(* CODESYS project sql_v_2_5_9.library
   DefaultNamespace: Teknike_SQL
   DocFormat: reStructuredText
   Description: Bliblioteca para controle do SQL usando todas as outras blibliotecas
   Author: Tiago B. Cunico
   Title: SQL
   Version: 2.5.9
   Company: Teknike
   Placeholder: Teknike_SQL

Project tree, tasks and I/O mapping:
  libraries: OSCAT - AixOCAT, * (RWTH Aachen University - E.ON Energy Research Center); Tc2_ModbusRTU, * (Beckhoff Automation GmbH); Tc2_Standard, * (Beckhoff Automation GmbH); Tc2_System, * (Beckhoff Automation GmbH); Tc2_Utilities, * (Beckhoff Automation GmbH); Tc3_Database, * (Beckhoff Automation GmbH); Tc3_Module, * (Beckhoff Automation GmbH); Geral, * (Teknike); Partidas, * (Teknike); Sensores, * (Teknike)
  FBs/
    Emergencias/
      function block FB_CriaTabelaEmergencias [ST]: GeraAsEmergencias, GeraTabela
      function block FB_IniciaOsBlocosDaEmergencia [ST]
    Grupos/
      Sts/
        data type ST_BancoGrupo
        data type st_ConfigGrupo
        data type st_EntradaGrupo
        data type st_Grupo
        data type st_SaidaGrupo
      function F_StringSeparadorFBGrupos [ST]
      function block FB_ControleGrupo [ST]: AjustaEntrada, AjustaSaida, GeraTabela, MaquinaDeEstado
      function block FB_IniciaGrupos [ST]: GeraOsGrupos, GeraTabela, MaquinaInica
    IHM/
      STs/
        data type st_OutrosInterlocks
      function block FB_GeraListaInterlocksIHM [ST]
    Iluminacao/
      Duts/
        data type ConfigTelerruptorDB
        data type enum_GravaNomes
        data type enum_LeituradosNomes
      function block FB_ConfigDoTelerruptor [ST]: GeraOsTelerruptores, GeraTabela, GravaValores, LeNomes
    Intralogistica/
      Top10SKU/
        data type DUT_Top10SKU
        data type Enum_HistorogramaSKUs
        function block FB_HistogramaSKUsMaisLidas [ST]: Evento, GeraTabela, Tabela, Top10
        TODO.txt
    MedicaoEnergia/
      Duts/
        PM2100_485_Schneider/
          data type config_PM2100_485_Schneider
          data type entrada_PM2100_485_Schneider
          data type saida_PM2100_485_Schneider
          data type st_PM2100_485_Schneider
          data type State_Modbus
          data type stCorrente
          data type stDemanda
          data type stEnergia
          data type stPotencia
          data type stTensao
        SEPAMS20_485_Schneider/
          data type config_SEPAMS20_Schneider
          data type entrada_SEPAMS20_Schneider
          data type saida_SEPAMS20_Schneider
          data type st_SEPAMS20_Schneider
          data type stCorrenteSEPAM
          data type stTemposSEPAM
          data type stTensaoSEPAM
        data type stCentroDeCusto
        data type stConfigNomeMedidorDB
        data type stCorrenteCSV
        data type stEscreveNoSQL
        data type stLeDoSQL
        data type stMedia15min
        data type stMediaAno
        data type stMediaDia
        data type stMediaMes
        data type stMinuto
        data type stOrganizaDados
      function block FB_CentroDeCustos2 [ST]: LeValores
      function block FB_DBCentroDeCustos [ST]: DeleteValores, GeraTabela, GravaValores, LeValores
      function block FB_DBMedidores [ST]: GeraTabela, GravaValores, LeValores
      function block FB_LeBancoDeDadosParaCSV [ST]: GeraTabela, LeValores
      function block FB_NomesMedidoresPM2100 [ST]: GeraOsMedidores, GeraTabela, GravaValores, LeNomes
      function block FB_NomesMedidoresSEPAM [ST]: GeraOsMedidores, GeraTabela, GravaValores, LeNomes
      function block FB_SalvaDadosMedidores [ST]: GeraTabela, GravaValores
    Partidas/
      KPI/
        function block FB_KPIPartidasSQL [ST]: GeraTabela, GravaHistorico
        data type st_KPISQL
      SalvaUsoNormal/
        function block FB_BDMotores [ST]: AtualizaValor, EscreveCSV, GeraTabela
        data type st_EscritaBD
      st/
        data type enum_MaquinaConfigPartidaDB
        data type st_LeConfigPartidaNoBanco_1
      function block FB_ConfigPartidaNoBanco [ST]: CalculaEmergencia, CalculaInterlock, ExecutaEstadoLeitura, GeraEmergencias, GeraNomeInterlock, LinkaOsNaoInterlock, MudouNoMotor, TrocaEstadoLeitura, ZeraReferencias
      function block FB_CriaTabelaEMotoresParaInterlock [ST]: GeraOsMotores, GeraTabela
      function block FB_IniciaOsBlocosDeConfigDoMotor [ST]: AtualizaTagEmergencias, AtualizaTagInterlocks, LinkaOsNaoInterlocks
    Sensores/
      fb_Hidrometro/
        dut/
          data type st_Hidrometro
        function block FB_Hidrometro [ST]: SalvaHistorico
      St/
        data type st_ComparaAnalogico
        data type st_LeComparaAnalogico
      function block FB_AtualizaTag [ST]: Atualiza, GeraTabela
      function block FB_CriaTabelaSensores [ST]: GeraOsSensores, GeraTabela
      function block FB_DBComparaSensor [ST]: GeraTabela, GravaValores
      function block FB_HistoricoSQL [ST]: GeraTabela, GravaHistorico
      function block FB_HistoricoTag [ST]: Atualiza, GeraTabela
      function block FB_IniciaOsBlocosDeSensor [ST]
    Valvula/
      BancoValvula/
  00000000-0000-0000-0000-000000000000|FBs\Intralogistica\Top10SKU\TODO.txt
  POUs/
    global variables GVL_BlibliotecaSQL
    program MAIN [ST]
    program ValidaLicensa [ST]: Licensas
  Project Information/
    function F_GetCompany [ST]
    function F_GetTitle [ST]
    function F_GetVersion [ST]
  Version/
    global variables Global_Version
  VISUs/
*)

// FBs/Grupos/Sts/ST_BancoGrupo
TYPE ST_BancoGrupo :
STRUCT
	ID: LINT;
	Nome: STRING(80);
	Motores: STRING(255);
	Timestamp: DT;
END_STRUCT
END_TYPE

// FBs/Grupos/Sts/st_ConfigGrupo
TYPE st_ConfigGrupo :
STRUCT PERSISTENT RETAIN
	sMotores: STRING(255);//se ele nao conseguir ler do banco ele pega daqui
	sNome : STRING;
	xCascata : BOOL;// assim ele usa cascata
	rTempoCascata : REAL; // ignora se a partida diz que ta show e liga por esse tempo
	xInterDependependes : BOOL; // se uma parar para todas
END_STRUCT
END_TYPE

// FBs/Grupos/Sts/st_EntradaGrupo
TYPE st_EntradaGrupo :
STRUCT
	xLiga : BOOL;
	xLigaFisico : BOOL;
	xReset : BOOL;
END_STRUCT
END_TYPE

// FBs/Grupos/Sts/st_Grupo
TYPE st_Grupo :
STRUCT
	En : st_EntradaGrupo;
	Sa : st_SaidaGrupo;
	Config : st_ConfigGrupo;
	Banco : ST_BancoGrupo;
END_STRUCT
END_TYPE

// FBs/Grupos/Sts/st_SaidaGrupo
TYPE st_SaidaGrupo :
STRUCT
	xError : BOOL;
	xInterlock : BOOL;
	xEmergencia : BOOL;
	xLigado : BOOL;
	xLigando : BOOL;
	sStatus : STRING;
	sStatusPartidas : ARRAY[0..100] OF STRING;
END_STRUCT
END_TYPE

// FBs/IHM/STs/st_OutrosInterlocks
TYPE st_OutrosInterlocks :
	STRUCT
		sTag	: STRING;
		xEstado	: BOOL;
	END_STRUCT
END_TYPE

// FBs/Iluminacao/Duts/ConfigTelerruptorDB
TYPE ConfigTelerruptorDB :
STRUCT
	Telerruptor: DINT;
	Tag: STRING(80);
	Funcao: STRING(80);
END_STRUCT
END_TYPE

// FBs/Iluminacao/Duts/enum_GravaNomes
{attribute 'qualified_only'}
{attribute 'strict'}
TYPE enum_GravaNomes :
(
	eEsperando := 0,
	eAbreConexao := 1,
	eGravaNomes := 2,
	eCriaComando := 3,
	eFechaConexao := 4,
	eParado := 100
);
END_TYPE

// FBs/Iluminacao/Duts/enum_LeituradosNomes
{attribute 'qualified_only'}
{attribute 'strict'}
TYPE enum_LeituradosNomes :
(
	eEsperando := 0,
	eAbreConexao := 1,
	eLeOsNomes := 2,
	eMonitoraTrocaDeNomes := 3,
	eFechaConexao := 4,
	eParado := 100
);
END_TYPE

// FBs/Intralogistica/Top10SKU/DUT_Top10SKU
TYPE DUT_Top10SKU :
STRUCT
	SKU : LINT;
	Contagem : LINT;
END_STRUCT
END_TYPE

// FBs/Intralogistica/Top10SKU/Enum_HistorogramaSKUs
{attribute 'qualified_only'}
//{attribute 'strict'}
TYPE Enum_HistorogramaSKUs :
(
	erro := 0,
	Esperando,
	AbreConexao,
	CriaComando,
	Grava,
	DeletaEvento,
	CriaEvento,
	Vetop10,
	FechaConexao
);
END_TYPE

// FBs/MedicaoEnergia/Duts/PM2100_485_Schneider/config_PM2100_485_Schneider
TYPE config_PM2100_485_Schneider :
STRUCT PERSISTENT RETAIN
	iEndereco 			: INT;
	sNomeFuncao			: STRING; 
END_STRUCT
END_TYPE

// FBs/MedicaoEnergia/Duts/PM2100_485_Schneider/entrada_PM2100_485_Schneider
TYPE entrada_PM2100_485_Schneider :
STRUCT
	xInicia				: BOOL; //Inicia a leitura
	xAtualizaCorrente	: BOOL := TRUE; //Habilita para ler os parametros de corrente
	xAtualizaTensao		: BOOL;	//Habilita para ler os parametros de tensao
	xAtualizaPotencia	: BOOL; //Habilita para ler os parametros de potencia
	xAtualizaEnergia	: BOOL := TRUE; //Habilita para ler os parametros de energia
	xAtualizaDemanda	: BOOL := TRUE; //Habilita para ler os parametros de demanda
END_STRUCT
END_TYPE

// FBs/MedicaoEnergia/Duts/PM2100_485_Schneider/saida_PM2100_485_Schneider
TYPE saida_PM2100_485_Schneider :
STRUCT
	xTerminei					: BOOL;	
	xOnline						: BOOL;
	UltimoModbusErro			: ST_ModbusErrorDiagnostics;
	sStatus						: STRING;
	Corrente: stCorrente;
	Tensao	: stTensao;
	Energia	: stEnergia;
	Potencia: stPotencia;
	Demanda	: stDemanda;
END_STRUCT
END_TYPE

// FBs/MedicaoEnergia/Duts/PM2100_485_Schneider/st_PM2100_485_Schneider
TYPE st_PM2100_485_Schneider :
STRUCT
	en		: entrada_PM2100_485_Schneider;
	sa		: saida_PM2100_485_Schneider;
	config	: config_PM2100_485_Schneider;
END_STRUCT
END_TYPE

// FBs/MedicaoEnergia/Duts/PM2100_485_Schneider/State_Modbus
{attribute 'qualified_only'}
{attribute 'strict'}
TYPE State_Modbus :
(
	Inicia			:= 0,
	LeituraCorrente	:= 1,
	LeituraTensao	:= 2,
	LeituraPotencia	:= 3,
	LeituraEnergia	:= 4,
	LeituraDemanda	:= 5,
	LeituraTempos	:= 6 
);
END_TYPE

// FBs/MedicaoEnergia/Duts/PM2100_485_Schneider/stCorrente
TYPE stCorrente :
STRUCT
	//Corrente
	rCorrenteA		: REAL;
	rCorrenteB		: REAL;
	rCorrenteC		: REAL;
	rCorrenteMedia	: REAL;
END_STRUCT
END_TYPE

// FBs/MedicaoEnergia/Duts/PM2100_485_Schneider/stDemanda
TYPE stDemanda :
STRUCT
	//Demanda
	rDemandaDePotenciaAtiva		: REAL;
	rDemandaDePotenciaReativa	: REAL;
	rDemandaDePotenciaAparente	: REAL;
END_STRUCT
END_TYPE

// FBs/MedicaoEnergia/Duts/PM2100_485_Schneider/stEnergia
TYPE stEnergia :
STRUCT
	//Energia
	rPotenciaAtivaEntregue		: REAL;
	rPotenciaAtivaRecebida		: REAL;
	rPotenciaReativaEntregue	: REAL;
	rPotenciaReativaRecebida	: REAL;
	rPotenciaAparenteEntregue	: REAL;
	rPotenciaAparenteRecebida	: REAL;
END_STRUCT
END_TYPE

// FBs/MedicaoEnergia/Duts/PM2100_485_Schneider/stPotencia
TYPE stPotencia :
STRUCT
	//Potencia
	rPotenciaAtivaTotal		: REAL;
	rPotenciaReativaTotal	: REAL;
	rPotenciaAparenteTotal	: REAL;
	rFatorDePotenciaTotal	: REAL;
END_STRUCT
END_TYPE

// FBs/MedicaoEnergia/Duts/PM2100_485_Schneider/stTensao
TYPE stTensao :
STRUCT
	//Tensao
	rTensaoAN		: REAL;
	rTensaoBN		: REAL;
	rTensaoCN		: REAL;
	rTensaoMediaLN	: REAL;
	rTensaoAB		: REAL;
	rTensaoBC		: REAL;
	rTensaoAC		: REAL;
	rTensaoMediaLL	: REAL;
END_STRUCT
END_TYPE

// FBs/MedicaoEnergia/Duts/SEPAMS20_485_Schneider/config_SEPAMS20_Schneider
TYPE config_SEPAMS20_Schneider :
STRUCT PERSISTENT RETAIN
	iEndereco 			: INT;
	sNomeFuncao			: STRING;
END_STRUCT
END_TYPE

// FBs/MedicaoEnergia/Duts/SEPAMS20_485_Schneider/entrada_SEPAMS20_Schneider
TYPE entrada_SEPAMS20_Schneider :
STRUCT
	xInicia				: BOOL; //Inicia a leitura
	xAtualizaCorrente	: BOOL := TRUE; //Habilita para ler os parametros de corrente
	xAtualizaTensao		: BOOL := TRUE;	//Habilita para ler os parametros de tensao
	xAtualizaTempos		: BOOL; //Habilita para ler os parametros que indicam tempos de atuação do disjuntor
END_STRUCT
END_TYPE

// FBs/MedicaoEnergia/Duts/SEPAMS20_485_Schneider/saida_SEPAMS20_Schneider
TYPE saida_SEPAMS20_Schneider :
STRUCT
	xTerminei					: BOOL;	
	xOnline						: BOOL;
	UltimoModbusErro			: ST_ModbusErrorDiagnostics;
	sStatus						: STRING;
	
	rDemandaAparente			: REAL;	
	Corrente					: stCorrenteSEPAM;
	Tensao						: stTensaoSEPAM;
	Tempos						: stTemposSEPAM;
END_STRUCT
END_TYPE

// FBs/MedicaoEnergia/Duts/SEPAMS20_485_Schneider/st_SEPAMS20_Schneider
TYPE st_SEPAMS20_Schneider :
STRUCT
	en		: entrada_SEPAMS20_Schneider;
	sa		: saida_SEPAMS20_Schneider;
	config	: config_SEPAMS20_Schneider;
END_STRUCT
END_TYPE

// FBs/MedicaoEnergia/Duts/SEPAMS20_485_Schneider/stCorrenteSEPAM
TYPE stCorrenteSEPAM :
STRUCT
	//Corrente
	rCorrente1		: REAL;
	rCorrente2		: REAL;
	rCorrente3		: REAL;
	rCorrente1Media	: REAL;
	rCorrente2Media	: REAL;
	rCorrente3Media	: REAL;
	rCorrenteTrip1	: REAL;
	rCorrenteTrip2	: REAL;
	rCorrenteTrip3	: REAL;
END_STRUCT
END_TYPE

// FBs/MedicaoEnergia/Duts/SEPAMS20_485_Schneider/stTemposSEPAM
TYPE stTemposSEPAM :
STRUCT
	iTempoDeOperacao					: INT;
	iTempoDeOperacaoAntesDoTrip			: INT;
	iTempoDeEsperaAposTripPorSobrecarga	: INT;
	iTempoDeInibicaoDePartida			: INT;
END_STRUCT
END_TYPE

// FBs/MedicaoEnergia/Duts/SEPAMS20_485_Schneider/stTensaoSEPAM
TYPE stTensaoSEPAM :
STRUCT
	rTensaoV1	: REAL;
	rTensaoV2	: REAL;
	rTensaoV3	: REAL;
	rTensaoU21	: REAL;
	rTensaoU32	: REAL;
	rTensaoU13	: REAL;
END_STRUCT
END_TYPE

// FBs/MedicaoEnergia/Duts/stCentroDeCusto
TYPE stCentroDeCusto :
STRUCT
	NomeGrupo				: STRING(255);
	MedidoresSelecionados	: STRING(255);
	Timestamp				: DT;
END_STRUCT
END_TYPE

// FBs/MedicaoEnergia/Duts/stConfigNomeMedidorDB
TYPE stConfigNomeMedidorDB :
STRUCT
	Medidor: DINT;
	Tag: STRING(80);
	Funcao: STRING(80);
END_STRUCT
END_TYPE

// FBs/MedicaoEnergia/Duts/stCorrenteCSV
TYPE stCorrenteCSV :
STRUCT
	rCorrenteA				: REAL;
	rCorrenteB				: REAL;
	rCorrenteC				: REAL;
	rCorrenteMedia			: REAL;
	Medidor					: INT;
	Timestamp				: DT;
END_STRUCT
END_TYPE

// FBs/MedicaoEnergia/Duts/stEscreveNoSQL
TYPE stEscreveNoSQL :
STRUCT
	rDemanda1min			: REAL;
	rFatorDePotencia1min	: REAL;
	rConsumo1min			: REAL;
	xTrocouMinuto			: BOOL;
END_STRUCT
END_TYPE

// FBs/MedicaoEnergia/Duts/stLeDoSQL
TYPE stLeDoSQL :
STRUCT
	Minuto		: ARRAY[1..15] OF stMinuto;
	Media15min	: ARRAY[1..96] OF stMedia15min;
	MediaDia	: ARRAY[1..31] OF stMediaDia;
	MediaMes	: ARRAY[1..12] OF stMediaMes;
END_STRUCT
END_TYPE

// FBs/MedicaoEnergia/Duts/stMedia15min
TYPE stMedia15min :
STRUCT
	rMedia15min				: REAL;
	rFatorDePotencia15min	: REAL;
	rConsumo15min			: REAL;
	Medidor					: INT;
	Timestamp				: DT;
END_STRUCT
END_TYPE

// FBs/MedicaoEnergia/Duts/stMediaAno
TYPE stMediaAno :
STRUCT
	rMediaAno			: REAL;
	rFatorDePotenciaAno	: REAL;
	rConsumoAno			: REAL;
	Medidor				: INT;
	Timestamp			: DT;
END_STRUCT
END_TYPE

// FBs/MedicaoEnergia/Duts/stMediaDia
TYPE stMediaDia :
STRUCT
	rMediaDia				: REAL;
	rFatorDePotenciaDia		: REAL;
	rConsumoDia				: REAL;
	Medidor					: INT;
	Timestamp				: DT;
END_STRUCT
END_TYPE

// FBs/MedicaoEnergia/Duts/stMediaMes
TYPE stMediaMes :
STRUCT
	rMediaMes			: REAL;
	rFatorDePotenciaMes	: REAL;
	rConsumoMes			: REAL;
	Medidor				: INT;
	Timestamp			: DT;
END_STRUCT
END_TYPE

// FBs/MedicaoEnergia/Duts/stMinuto
TYPE stMinuto :
STRUCT
	rDemanda1min		: REAL;
	rFatorDePotencia1min: REAL;
	rConsumo1min		: REAL;
	Medidor				: INT;
	Timestamp			: DT;
END_STRUCT
END_TYPE

// FBs/MedicaoEnergia/Duts/stOrganizaDados
TYPE stOrganizaDados :
STRUCT
	iMedidor	: INT;
	minuto		: ARRAY[1..15] OF stMinuto;
	media15min	: ARRAY[1..96] OF stMedia15min;
	MediaDia	: ARRAY[1..31] OF stMediaDia;
	MediaMes	: ARRAY[1..12] OF stMediaMes;
END_STRUCT
END_TYPE

// FBs/Partidas/KPI/st_KPISQL
TYPE st_KPISQL :
STRUCT
	ID : T_ULARGE_INTEGER;
	TAG : STRING;
	Desligado : REAL;
	Ligado : REAL;
	Emergencia : REAL;
	Falha : REAL;
	Interlock : REAL;
	//Timestamp : DT;
END_STRUCT
END_TYPE

// FBs/Partidas/SalvaUsoNormal/st_EscritaBD

TYPE st_EscritaBD :
	STRUCT
		ID					: T_ULARGE_INTEGER;
		Velocidade			: INT;
		Corrente			: REAL;
		TemperaturaDoMotor	: REAL;
		Torque				: REAL;
		StatusIHM			: STRING;
		HorimetroD			: STRING;
		TotalDePartidas		: INT;
		TotalDeFalhas		: INT;
	END_STRUCT
END_TYPE

// FBs/Partidas/st/enum_MaquinaConfigPartidaDB
{attribute 'qualified_only'}
{attribute 'strict'}
TYPE enum_MaquinaConfigPartidaDB :
(
	Esperando := 0,
	AbreConexao,
	CriaComando,
	Gravando,
	FechaConexao,
	LendoEleMesmo,
	LinkaOsNaoInterlock,
	ProcuraTag1,
	ProcuraTag2,
	Gera_sInterlock,
	Gera_Emergencia,
	ExecutaInterlocks,
	falha
);
END_TYPE

// FBs/Partidas/st/st_LeConfigPartidaNoBanco_1
TYPE ST_ConfigMotorDB_1 :
	STRUCT
		Motor	: T_ULARGE_INTEGER;
		Tag		: STRING(80);
		Funcao	: STRING(80);

		InvIT1A	: INT;
		IT1A	: STRING(80);
		OPIT1	: INT;
		InvIT1B	: INT;
		IT1B	: STRING(80);

		InvIT2A	: INT;
		IT2A	: STRING(80);
		OPIT2	: INT;
		InvIT2B	: INT;
		IT2B	: STRING(80);

		InvIT3A	: INT;
		IT3A	: STRING(80);
		OPIT3	: INT;
		InvIT3B	: INT;
		IT3B	: STRING(80);

		InvIT4A	: INT;
		IT4A	: STRING(80);
		OPIT4	: INT;
		InvIT4B	: INT;
		IT4B	: STRING(80);
		
		Timestamp : DT;

	END_STRUCT
END_TYPE

// FBs/Sensores/fb_Hidrometro/dut/st_Hidrometro
TYPE st_Hidrometro :
STRUCT
	rContadorTotal : REAL;
	rContadorHoje : REAL;
	xSinal : BOOL;
	xReset : BOOL;
	Historico : ARRAY[0..180] OF st_HistoricoHidrometro;
	rMultiplicadorVazao : REAL := 0.1;
END_STRUCT
END_TYPE

// FBs/Sensores/St/st_ComparaAnalogico
TYPE st_ComparaAnalogico :
STRUCT
	rAnalogicoLido	: REAL;
	rAnalogicoManual: REAL;
	rDiferenca		: REAL;
	xSalva			: BOOL;
END_STRUCT
END_TYPE

// FBs/Sensores/St/st_LeComparaAnalogico
TYPE st_LeComparaAnalogico :
	STRUCT
		Sensor			: T_ULARGE_INTEGER;
		rAnalogicoLido	: REAL;
		rAnlogicoManual	: REAL;
		rDiferenca		: REAL;
		xSalva			: BOOL;
	END_STRUCT
END_TYPE

// POUs/GVL_BlibliotecaSQL
//{attribute 'qualified_only'}
VAR_GLOBAL
    {attribute 'hide'} 
	{attribute 'tc_no_symbol'}
	xLicensaValida651641iih : BOOL;
	LicensaValida : BOOL;
	STCheckLicense : ST_CheckLicense;
END_VAR

// Version/Global_Version
{attribute 'TcGenerated'}
{attribute 'no-analysis'}
{attribute 'linkalways'}
// This function has been automatically generated from the project information.
VAR_GLOBAL CONSTANT
	{attribute 'const_non_replaced'}
	stLibVersion_SQL : ST_LibVersion := (iMajor := 2, iMinor := 5, iBuild := 9, iRevision := 0, nFlags := 0, sVersion := '2.5.9');
END_VAR

// FBs/Emergencias/FB_CriaTabelaEmergencias
(*
	Bloco para gerar a tabela das emergencias de forma generica
*)


{attribute 'hide_all_locals'}
FUNCTION_BLOCK FB_CriaTabelaEmergencias
VAR_IN_OUT
	Emergencias : ARRAY[*] OF st_Emergencia;
END_VAR
VAR_INPUT
	xCriaTabela		: BOOL;
	iNumeroDataBase	: INT		:= 1;
	sNomeDataBase	: STRING	:= 'EmergenciaConfig';
END_VAR
VAR_OUTPUT
	xOcupado : BOOL;
END_VAR
VAR
	i				: INT;
	xGeraMoto		: BOOL;
	diParteBaixa	: DINT;
	diParteAlta		: DINT;

	//Grava valores
	xGravando		: BOOL;
	rtEscrita		: R_TRIG;
	xEscreve		: BOOL;
	EstruturaBanco	: st_Emergencia_Banco;
	xEscreveAux		: BOOL;
	sAux			: ARRAY[1..50] OF STRING(80);
	fbPLCDBWrite	: FB_PLCDBWriteEvt(sNetID := '', tTimeout := T#30S); //Bloco para gravar no banco de dados

	ColumnNamesGrava : ARRAY[0..2] OF STRING(50) := ['Emergencia',
													'Tag',
													'Funcao'];

	//Cria table
	rtCria			: R_TRIG;
	xCria			: BOOL;
	fbPLCDBCreate	: FB_PLCDBCreateEvt(sNetID := '', tTimeout := T#30S);

	ColumnInfo :
		ARRAY[0..3] OF ST_ColumnInfo
		:= [(sName := 'Emergencia', eType := E_ColumnType.BigInt, nLength := 8, sProperty := 'IDENTITY(1,1)'),
				(sName := 'Tag', eType := E_ColumnType.NVarChar, nLength := 80, sProperty := 'DEFAULT $'SEMTAG$''),
				(sName := 'Funcao', eType := E_ColumnType.NVarChar, nLength := 80, sProperty := 'DEFAULT $'NADA$''),
				(
				sName := 'Timestamp',
					eType := E_ColumnType.DateTime,
					nLength := 4,
					sProperty := 'DEFAULT CURRENT_TIMESTAMP ON UPDATE CURRENT_TIMESTAMP')];
END_VAR

IF xLicensaValida651641iih THEN
	GeraTabela();
	GeraAsEmergencias();
END_IF

ACTION GeraAsEmergencias:

diParteBaixa	:= LOWER_BOUND(Emergencias, 1);
diParteAlta		:= UPPER_BOUND(Emergencias, 1);

IF xGeraMoto THEN

	xEscreve := TRUE;
	rtEscrita(CLK := xEscreve, Q =>);

	IF rtEscrita.q THEN
		xEscreveAux						:= TRUE;
		//EstruturaBanco.Sensor.dwLowPart	:= DINT_TO_DWORD(diParteBaixa + i);
		EstruturaBanco.Tag				:= CONCAT('Emer', TO_STRING(i));
	END_IF

	IF xEscreveAux THEN
		IF fbPLCDBWrite.WriteStruct
			(
				hDBID := INT_TO_UDINT(iNumeroDataBase),
					sTableName := sNomeDataBase,
					pRecord := ADR(EstruturaBanco),
					cbRecord := SIZEOF(EstruturaBanco),
					pColumnNames := ADR(ColumnNamesGrava),
					cbColumnNames := SIZEOF(ColumnNamesGrava))
		THEN
			xEscreve := FALSE;
			rtEscrita(CLK := xEscreve, Q =>);
			xEscreveAux	:= FALSE;
			i			:= i + 1;

			IF i > diParteAlta THEN
				xGeraMoto	:= FALSE;
				xOcupado	:= FALSE;
			END_IF
		END_IF
	END_IF

END_IF
END_ACTION

ACTION GeraTabela:

rtCria(CLK := xCriaTabela, Q =>);

IF rtCria.q THEN
	xCria		:= TRUE;
	xOcupado	:= TRUE;
END_IF

IF xCria THEN

	IF fbPLCDBCreate.Table
		(
			hDBID := INT_TO_UDINT(iNumeroDataBase),
				sTableName := sNomeDataBase,
				pTableCfg := ADR(ColumnInfo),
				cbTableCfg := SIZEOF(ColumnInfo))
	THEN
		IF NOT fbPLCDBCreate.bError THEN
			xCria		:= FALSE;
			xCriaTabela	:= FALSE;
			xGeraMoto	:= TRUE;
			i			:= 1;
		ELSE
			xCria		:= FALSE;
			xCriaTabela	:= FALSE;
		END_IF
	END_IF

END_IF
END_ACTION

END_FUNCTION_BLOCK

// FBs/Emergencias/FB_IniciaOsBlocosDaEmergencia
{attribute 'hide_all_locals'}
FUNCTION_BLOCK FB_IniciaOsBlocosDaEmergencia
VAR_IN_OUT
	stEmergencias : ARRAY[*] OF st_Emergencia;
	sPossiveisEmergencias : ARRAY[*] OF STRING;
END_VAR
VAR_INPUT
	xInicia : BOOL;
	iNumeroDataBase	: INT		:= 1;
	sNomeDataBase	: STRING	:= 'EmergenciaConfig';
END_VAR
VAR_OUTPUT
END_VAR
VAR
	fbPLCDBCmd			: FB_PLCDBCmdEvt(sNetID := '', tTimeout := T#60S);
	fbSQLDatabase		: FB_SQLDatabaseEvt(sNetID := '', tTimeout := T#60S);
	sCmd				: STRING(1000);
	sCmdUpdate			: STRING(1000);
	stPara				: ST_ExpParameter;
	TagAProcurar		: STRING(80);
	nRecords			: UDINT;
	xProcuraNaTabela	: BOOL;
	EstruturaBanco		: ARRAY[0..999] OF Teknike_Geral.st_Emergencia_Banco;
	xJogaNoInterlock	: BOOL;
	sTag1				: STRING;
	sTag2				: STRING;
	xEMotor				: BOOL;
	sMensagemErro1		: STRING;
	diCimaSensor		: DINT;
	diBaixoSensor		: DINT;

	iEstado	: INT := 1;
	i		: INT;

	iAux : INT;
	
	EstruturaBancoVazio: Teknike_Geral.st_Emergencia_Banco;

END_VAR


IF xLicensaValida651641iih THEN
	
	
	CASE iEstado OF
		1: //Esperando
			IF xInicia THEN
				iEstado := 2;
			END_IF
	
		2: //abre conexao
			IF fbSqlDatabase.Connect(int_to_udint(iNumeroDataBase)) THEN
				IF fbSqlDatabase.bError THEN
					IF fbSqlDatabase.ipTcResult.ipSourceInfo.sName = 'ADSERR_DEVICE_LICENSENOTFOUND' THEN
						// se der isso ele nao fica tentando e gerando uma caralhada de erro pq nao tem a lisença
						iEstado := 0;
					ELSE
						iEstado := 2;
					END_IF
				ELSE
					IF fbSqlDatabase.bConnected THEN
						iEstado := 3;
					END_IF
				END_IF
			END_IF
	
		3: // le o role
			TagAProcurar		:= sTag1;
			stPara.eParaType	:= E_ExpParameterType.STRING_;
			stPara.nParaSize	:= SIZEOF(TagAProcurar);
			stPara.sParaName	:= 'Tag';
	
			diBaixoSensor	:= LOWER_BOUND(stEmergencias, 1);
			diCimaSensor	:= UPPER_BOUND(stEmergencias, 1);
	
			// set command with placeholder
			sCmd := CONCAT(CONCAT('SELECT * FROM ',sNomeDataBase),';');
	
			// call functionblock
			IF fbPLCDBCmd.ExecuteDataReturn
				(
					hDBID := 1,
						pExpression := ADR(sCmd),
						cbExpression := SIZEOF(sCmd),
						pData := ADR(TagAProcurar),
						cbData := SIZEOF(TagAProcurar),
						pParameter := ADR(stPara),
						cbParameter := SIZEOF(stPara),
						nStartIndex := 0,
						nRecordCount := DINT_TO_UDINT(diCimaSensor-1),
						pReturnData := ADR(EstruturaBanco),
						cbReturnData := SIZEOF(EstruturaBanco),
						pRecords := ADR(nRecords))
			THEN
				IF fbPLCDBCmd.bError THEN
					sMensagemErro1 := 'Nao conseguiu a tag';
				ELSE
					sMensagemErro1	:= 'Conseguiu a tag';
					iEstado			:= 4;
					
					//Fica forçado pra poder ter uma emergencia geral, tipo juntar varias numa
					IF diBaixoSensor = 0 THEN
						stEmergencias[0].Banco.Tag := 'Emergencia Geral';
					END_IF
	
					FOR i := TO_INT(diBaixoSensor) TO TO_INT(diCimaSensor)-1 DO
						stEmergencias[i+1].Banco := EstruturaBanco[i];
					END_FOR
					//Essa aqui fica vazia so pro framework aceitar colocar vazio
					stEmergencias[diCimaSensor].Banco := EstruturaBancoVazio;
				END_IF
			END_IF
	
		4: // FechaConexao conexao
			IF fbSqlDatabase.Disconnect() THEN
	
				xInicia := FALSE;
	
				IF fbSqlDatabase.bError THEN
					iEstado := 1;
				ELSE
					iEstado := 1;
				END_IF
				
				//IF LOWER_BOUND(sPossiveisEmergencias,1) = LOWER_BOUND(stEmergencias,1) AND UPPER_BOUND(sPossiveisEmergencias,1)+1 = UPPER_BOUND(stEmergencias,1) THEN	
					FOR i:= TO_INT(LOWER_BOUND(sPossiveisEmergencias,1)) TO TO_INT(UPPER_BOUND(sPossiveisEmergencias,1)) DO
						sPossiveisEmergencias[i] := stEmergencias[i].Banco.Tag;
					END_FOR
				//ELSE
				//	sPossiveisEmergencias[LOWER_BOUND(sPossiveisEmergencias,1)] := 'Vetor de tamanho errado';
				//END_IF
				
				
			END_IF
	END_CASE

END_IF

END_FUNCTION_BLOCK

// FBs/Grupos/F_StringSeparadorFBGrupos
FUNCTION F_StringSeparadorFBGrupos : BOOL
VAR_INPUT
	sStr : STRING;
END_VAR
VAR_IN_OUT
	ListaINT : ARRAY[*] OF INT;
END_VAR
VAR
	iListIntMIN : INT;
	iListIntMAX : INT;
	
	sParteEsquerda : STRING;
	sResto : STRING;
	sSepara : STRING;
	
	sNumeroInicio : STRING;
	sNumeroFim : STRING;
	
	i: INT;
	j: INT;
	
	iIndex : INT;
END_VAR


iListIntMIN := DINT_TO_INT(LOWER_BOUND(ListaINT,1));
iListIntMAX := DINT_TO_INT(UPPER_BOUND(ListaINT,1));

FOR i:= iListIntMIN TO iListIntMAX DO
	ListaINT[i] := 0;
END_FOR


sSepara := sStr;
iIndex := iListIntMIN;

//O codigo aqui vai pegar a string que a gente guarda no banco de dados e separar onde tem ","
//quando ele separa ele ve se dentro ta um "-", que nesse caso esta servindo para colocar os motores dentro de um periodo
// entao se se ele revceber a string 1-5,7,10 ele devolver na lista os motores do 1,2,3,4,5,7,10
//ele olha tb ser nao entrou um motor 2 vezes, se for o caso ele considera so a primeira vez

WHILE FindAndSplit(
		pSeparator:= ADR(','), 
		pSrcString:= ADR(sSepara), 
		pLeftString:= ADR(sParteEsquerda), 
		nLeftSize:= SIZEOF(sParteEsquerda), 
		pRightString:= ADR(sResto), 
		nRightSize:= SIZEOF(sResto), 
		bSearchFromRight:= FALSE) DO
	
	IF FIND(STR1:= sParteEsquerda, STR2:='-' ) = 0 THEN// se nao tem o "-" 	
		FOR i := 1 TO iIndex DO
			IF ListaINT[i] = STRING_TO_INT(sParteEsquerda) THEN	
				EXIT;
			END_IF
		END_FOR	
		IF i > iIndex THEN	
			ListaINT[iIndex]:= STRING_TO_INT(sParteEsquerda);
			iIndex := iIndex + 1;
		END_IF
	ELSE
		
		FindAndSplit(pSeparator:= ADR('-'),	pSrcString:= ADR(sParteEsquerda),
					 pLeftString:= ADR(sNumeroInicio), nLeftSize:= SIZEOF(sNumeroInicio), 
					 pRightString:= ADR(sNumeroFim), nRightSize:= SIZEOF(sNumeroFim), 
					 bSearchFromRight:= FALSE);
					
		FOR i := STRING_TO_INT(sNumeroInicio) TO STRING_TO_INT(sNumeroFim) DO
			FOR j := i TO iIndex DO
				IF ListaINT[j] = i THEN	
					EXIT;
				END_IF
			END_FOR	
			IF j > iIndex THEN	
				ListaINT[iIndex]:= i;
				iIndex := iIndex + 1;
			END_IF
		END_FOR
	
	
	END_IF
	sSepara := sResto;
	
	IF iIndex > iListIntMAX THEN
		F_StringSeparadorFBGrupos := FALSE;
		EXIT;
	END_IF
	
END_WHILE


// pega se so tem motores em sequencia sem um ','
IF FIND(STR1:= sSepara, STR2:='-' ) > 0 THEN
	
	FindAndSplit(pSeparator:= ADR('-'),	pSrcString:= ADR(sSepara),
				 pLeftString:= ADR(sNumeroInicio), nLeftSize:= SIZEOF(sNumeroInicio), 
				 pRightString:= ADR(sNumeroFim), nRightSize:= SIZEOF(sNumeroFim), 
				 bSearchFromRight:= FALSE);
					
		FOR i := STRING_TO_INT(sNumeroInicio) TO STRING_TO_INT(sNumeroFim) DO
			FOR j := 1 TO iIndex DO
				IF ListaINT[j] = i THEN	
					EXIT;
				END_IF
			END_FOR	
			IF j > iIndex THEN	
				ListaINT[iIndex]:= i;
				iIndex := iIndex + 1;
			END_IF
		END_FOR
		// joga vazio pra nao pegar no de baixo
		sSepara := '';
		sResto := '';
END_IF


FOR i := 1 TO iIndex DO
	IF ListaINT[i] = STRING_TO_INT(sSepara) THEN	
		EXIT;
	END_IF
END_FOR	
IF i > iIndex THEN	
	ListaINT[iIndex]:= STRING_TO_INT(sSepara);
END_IF



F_StringSeparadorFBGrupos := TRUE;

END_FUNCTION

// FBs/Grupos/FB_ControleGrupo
FUNCTION_BLOCK FB_ControleGrupo
VAR_IN_OUT
	stGrupo : st_Grupo;
	Motores : ARRAY[*] OF st_Partida;
END_VAR
VAR_INPUT
	iIndexGrupo : INT;
	iNumeroDataBase : INT := 1;
	sNomeTabela : STRING := 'GruposConfig';
	xLiga : BOOL;
	xLigaFisico : BOOL;
	xReset : BOOL;
	xAtualizaExternoErro : BOOL;
	iEstado : INT := -1;
	EstruturaBanco 	: ST_BancoGrupo; 
END_VAR
VAR_OUTPUT
	xError : BOOL;
	xLigado : BOOL;
	xLigando: BOOL;
	xInterlock : BOOL;
	xEmergencia : BOOL;
	sStatus : STRING;
END_VAR
VAR
	//Controle Geral
	iMotores : ARRAY[0..100] OF INT;
	stGrupoAnterior : st_Grupo;
	i : INT;
	
	
	// Estado 2
	fbCascata : FB_Cascata;
	xCascata : ARRAY[0..100] OF BOOL;
	
	//Estado 3
	xMudouMotores : BOOL;
	sAux : ARRAY[0..50] OF STRING(80);
	sCmdUpdate : STRING(1000);
	fbPLCDBCmd    : FB_PLCDBCmdEvt(sNetID := '', tTimeout := T#5S);
	aPara : ST_ExpParameter;
	
	
	//Estado 0
	fbPLCDBRead		: FB_PLCDBReadEvt(sNetID := '', tTimeout := T#30S); //Bloco para leitura do banco de dados sem filtro
	ColumnNamesLe 	: ARRAY[0..3] OF STRING(50) := ['ID',
													'Nome',
													'Motores',
													'Timestamp'];
	
	
	//Criar a tabela												
	rtCria : R_TRIG;
	xCriaTabela : BOOL;
	xCria : BOOL;
	fbPLCDBCreate	: FB_PLCDBCreateEvt(sNetID := '', tTimeout := T#30S);

		ColumnInfo : ARRAY[0..3] OF ST_ColumnInfo := [(sName := 'ID', eType := E_ColumnType.BigInt, nLength := 8, sProperty := 'IDENTITY(1,1)'),
												(sName := 'Nome', eType := E_ColumnType.NVarChar, nLength := 80),
												(sName := 'Motores', eType := E_ColumnType.NVarChar, nLength := 255),
												(
				sName := 'Timestamp',
					eType := E_ColumnType.DateTime,
					nLength := 4,
					sProperty := 'DEFAULT CURRENT_TIMESTAMP ON UPDATE CURRENT_TIMESTAMP')];


	sAuxEstado : STRING;
	
	xFirstScan : BOOL := TRUE;
	
	xInvalido : BOOL;
	chAux : STRING(1);
	
	rxAux : REFERENCE TO BOOL;
	xAux : BOOL;
	iAux : INT;
	
	
	btxLigaIHM : B_TRIG;
	
 
END_VAR



IF xLicensaValida651641iih THEN
	AjustaEntrada();
	GeraTabela();
	
	MaquinaDeEstado();
	AjustaSaida();
ELSE	
	ValidaLicensa();
END_IF





xFirstScan := FALSE;

ACTION AjustaEntrada:




IF stGrupo.en.xLiga <> stGrupoAnterior.en.xLiga THEN
	xliga := stGrupo.en.xLiga;
END_IF
IF stGrupo.en.xLiga <> xLiga THEN
	stGrupo.en.xLiga := xLiga;
END_IF

IF stGrupo.en.xLigaFisico <> stGrupoAnterior.en.xLigaFisico THEN
	xLigaFisico := stGrupo.en.xLigaFisico;
END_IF
IF stGrupo.en.xLigaFisico <> xLigaFisico THEN
	stGrupo.en.xLigaFisico := xLigaFisico;
END_IF


IF stGrupo.en.xReset <> stGrupoAnterior.en.xReset THEN
	xReset := stGrupo.en.xReset;
END_IF
IF stGrupo.en.xReset <> xReset THEN
	stGrupo.en.xReset := xReset;
END_IF



//aqui ele verifica se a string é valida
//se nao for ele volta o valor antigo pra ela
//ele olha pela tabela ascii, entao pode ter somente os caracteres
//2C,2d,30-39
IF stGrupo.Config.sMotores <> stGrupoAnterior.Config.sMotores THEN
	
	xInvalido := FALSE;

	IF F_StringIsASCII(ADR(stGrupo.Config.sMotores)) THEN
		
		FOR i:= 16#21 TO 16#7E DO
			IF NOT ((i >= 16#30 AND i <= 16#39) OR i = 16#2C OR i = 16#2D) THEN
				chAux := F_ToCHR(INT_TO_BYTE(i));
				IF FIND(STR1:= stGrupo.Config.sMotores, STR2:= chAux) > 0 THEN
					xInvalido := TRUE;
					EXIT;
				END_IF
			END_IF
		END_FOR
	END_IF
	
	IF xInvalido THEN
		stGrupo.Config.sMotores := stGrupoAnterior.Config.sMotores;
	ELSE
		xMudouMotores := TRUE;
	END_IF
END_IF
IF stGrupo.Config.sNome <> stGrupoAnterior.Config.sNome THEN
	xMudouMotores := true;
END_IF


stGrupoAnterior := stGrupo;
END_ACTION

ACTION AjustaSaida:


IF xFirstScan THEN
	FOR i := 0 TO 100 DO
		stGrupo.Sa.sStatusPartidas[i] := '-1';
	END_FOR
END_IF


xError := FALSE;
xInterlock := FALSE;
xEmergencia := FALSE;
FOR i := 0 TO 100 DO
	IF iMotores[i] = 0 THEN
		EXIT;
	END_IF
	xError := xError OR Motores[iMotores[i]].Sa.xFalha;
	xInterlock := xInterlock OR Motores[iMotores[i]].Sa.xParadoPorInterlock;
	xEmergencia := xEmergencia OR NOT Motores[iMotores[i]].En.xEmergenciaOK;
	iAux := iMotores[i];
	CASE Motores[iAux].Sa.iStsMotor OF
		0 :		sAuxEstado := ' - Bloco não esta rodando';
		1 :		sAuxEstado := ' - Parado em automatico';
		2 :		sAuxEstado := ' - Parado em manual';
		3 :		sAuxEstado := ' - Ligado em automatico';
		4 :		sAuxEstado := ' - Ligado em manual';
		5 :		sAuxEstado := ' - Bloqueado';
		6 :		sAuxEstado := ' - Falha contatora';
		7 :		sAuxEstado := ' - Inversor offline';
		8 :		sAuxEstado := ' - Disjuntor desarmado';
		9 :		sAuxEstado := ' - Emergencia';
		10 :	sAuxEstado := ' - Interlock';
		11 :	sAuxEstado := ' - Trocando sentido';
		12 :	sAuxEstado := ' - Inverosr em falha';
		13 :	sAuxEstado := ' - Falha freio';
		14 :	sAuxEstado := ' - Falha contato ok inversor';
		15 :	sAuxEstado := ' - Falha Soft';
		16 :	sAuxEstado := ' - Falha contato soft';
		17 :	sAuxEstado := ' - Higienização desligada';
		18 :	sAuxEstado := ' - Higienização ligada';
	END_CASE
	
	stGrupo.Sa.sStatusPartidas[i] := CONCAT(CONCAT(Motores[iAux].BancoDeDados.Tag,''),sAuxEstado);
	
END_FOR		



stGrupo.Sa.xError := xError;
stGrupo.Sa.xInterlock := xInterlock;
stGrupo.Sa.xEmergencia := xEmergencia;
stGrupo.Sa.xLigado := xLigado;
stGrupo.Sa.xLigando := xLiga AND NOT xligado;

IF xLiga AND NOT xligado THEN
	sStatus := 'Ligando';
ELSIF xLiga AND xligado THEN
	sStatus := 'Ligado';
ELSIF NOT xliga THEN
	sStatus := 'Desligado';
END_IF

IF xError THEN
	sStatus := CONCAT(sStatus,', Falha');
END_IF

stGrupo.Sa.sStatus := sStatus;
END_ACTION

ACTION GeraTabela:

rtCria(CLK := xCriaTabela, Q =>);

IF rtCria.q THEN
	xCria := TRUE;
END_IF

IF xCria THEN
	IF fbPLCDBCreate.Table(
			hDBID := INT_TO_UDINT(iNumeroDataBase),
			sTableName := sNomeTabela,
			pTableCfg := ADR(ColumnInfo),
			cbTableCfg := SIZEOF(ColumnInfo))
	THEN
		xCria := FALSE;
		xCriaTabela := FALSE;
	END_IF

END_IF
END_ACTION

ACTION MaquinaDeEstado:


CASE iEstado OF 
	0 : //Le Ele mesmo no banco
		IF fbPLCDBRead.ReadStruct(
								hDBID:=1 , 
								sTableName:= sNomeTabela, 
								pColumnNames:= ADR(ColumnNamesLe), 
								cbColumnNames:= SIZEOF(ColumnNamesLe), 
								sOrderByColumn:= ColumnNamesLe[0], 
								eOrderType:= E_OrderType.ASC, 
								nStartIndex:= iIndexGrupo-1, 
								nRecordCount:= 1, 
								pData:= ADR(EstruturaBanco), 
								cbData:= SIZEOF(EstruturaBanco))
		THEN
			iEstado := 1;	
		END_IF
		
	1 : // Atualiza Valores
		IF fbPLCDBRead.bError OR xAtualizaExternoErro THEN
			{error <'Não conseguiu ler ele mesmo no banco no bloco FB_ControleGrupo'>}
			
			//Se nao deu usa o que ja tem na memoria e vai com isso
			F_StringSeparadorFBGrupos(sStr:= stGrupo.config.sMotores, ListaINT:= iMotores);
			iEstado := 2;
			
		ELSE	
			//Ajeita o que veio do banco pra liberar o controle
			stGrupo.Banco := EstruturaBanco;
			stGrupo.Config.sMotores := EstruturaBanco.Motores;
			stGrupo.Config.sNome := EstruturaBanco.Nome;
			stGrupoAnterior := stGrupo;
			F_StringSeparadorFBGrupos(sStr:= EstruturaBanco.Motores, ListaINT:= iMotores);
			iEstado := 2;
		END_IF
		
		FOR i := 0 TO 100 DO
			stGrupo.Sa.sStatusPartidas[i] := '-1';
		END_FOR		
		
		xAtualizaExternoErro := FALSE;
		
		
	2 : // Esperando comando de liga ou pra atualizar a tabela
	
		IF xMudouMotores THEN
			iEstado := 3;
			xLiga := FALSE;
		END_IF
		
		//RESET
		IF xReset THEN
			FOR i := 0 TO 100 DO
				IF iMotores[i] = 0 THEN
					EXIT;
				END_IF
				Motores[iMotores[i]].En.xReset := TRUE;
			END_FOR
			xReset := FALSE;
		END_IF
		
		btxLigaIHM(CLK:= xLigaFisico, Q=> );
		IF btxLigaIHM.q THEN
			xLiga := xLigaFisico;
		END_IF
		
		xLigado := xLiga;
		
		// LIGA E DESLIGA
		IF xLiga THEN
			FOR i := 0 TO 100 DO
				IF iMotores[i] = 0 THEN
					EXIT;
				END_IF
				// Tem que ter uma condição la fora que jogue o xligaauto pra false
				IF NOT stGrupo.config.xCascata THEN	
					Motores[iMotores[i]].En.xLigaAuto := Motores[iMotores[i]].En.xLigaAuto OR TRUE;
				ELSE		
					Motores[iMotores[i]].En.xLigaAuto := Motores[iMotores[i]].En.xLigaAuto OR xCascata[i];
				END_IF
				
				xAux := Motores[iMotores[i]].En.xLigaAuto;
				
				xLigado := xLigado AND xAux;
				
			END_FOR
		END_IF
		
		fbCascata(	tCascata:= REAL_TO_TIME(stGrupo.Config.rTempoCascata*1000), 
					xLiga:= xLiga OR xLigaFisico, 
					xCascata:= xCascata, 
					iProximoALigar=> , 
					xLigado=> );
		
		
	3 : // manda pro banco os novos motores	
	
	
		xMudouMotores := FALSE;
	
		sAux[0] := CONCAT(CONCAT('UPDATE geral.',sNomeTabela),' SET ');

		sAux[1]	:= 'Nome = $'';
		sAux[2]	:= CONCAT((stGrupo.Config.sNome), '$', ');

		sAux[3]		:= 'Motores = $'';
		sAux[4]		:= (stGrupo.Config.sMotores);
		
		sAux[5]	:= '$' WHERE (ID = $'';
		sAux[6]	:= INT_TO_STRING(iIndexGrupo);
		sAux[7]	:= '$');';
		sCmdUpdate	:= F_ConcatArray1000(sArray := sAux);
		
		aPara.eParaType := E_ExpParameterType.STRING_;
		aPara.nParaSize := SIZEOF(sAux[0]);
		
		IF fbPLCDBCmd.Execute(
			hDBID:= 1, 
			pExpression:= ADR(sCmdUpdate), 
			cbExpression:= SIZEOF(sCmdUpdate), 
			pData:= ADR(sAux[0]), 
			cbData:= SIZEOF(sAux[0]), 
			pParameter:= ADR(aPara), 
			cbParameter:= SIZEOF(aPara))
		THEN
			iEstado := 0;
		END_IF
		
END_CASE
END_ACTION

END_FUNCTION_BLOCK

// POUs/ValidaLicensa
PROGRAM ValidaLicensa
VAR
{attribute 'tc_no_symbol'}
Olhaliscensa : FB_CheckLicense;
{attribute 'tc_no_symbol'}
GUIDLicensa : GUID := STRING_TO_GUID('7B4694D5-AEB4-4168-B911-6F1BA4CB3B1D');
END_VAR


Licensas();

STCheckLicense := Olhaliscensa.stCheckLicense;

xLicensaValida651641iih :=
 Olhaliscensa.stCheckLicense.eResult = 0 OR// essa é so pros que sao da beckhoff mesmo
 Olhaliscensa.stCheckLicense.eResult = 16#203 OR
 Olhaliscensa.stCheckLicense.eResult = 16#254 OR
 Olhaliscensa.stCheckLicense.eResult = 16#255;

 LicensaValida := xLicensaValida651641iih;

ACTION Licensas:
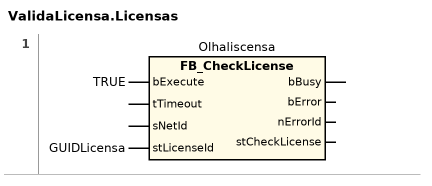
// NETWORK 1
Olhaliscensa(bExecute := TRUE, stLicenseId := GUIDLicensa); // FB_CheckLicense
END_ACTION

END_PROGRAM

// FBs/Grupos/FB_IniciaGrupos
FUNCTION_BLOCK FB_IniciaGrupos
VAR_INPUT
	xCriaTabela : BOOL;
	iNumeroDataBase : INT := 1;
	sNomeTabela : STRING := 'GruposConfig';
	xInicia : BOOL;
END_VAR
VAR_IN_OUT
	fbGrupos : ARRAY[*] OF FB_ControleGrupo;
END_VAR
VAR_OUTPUT
	xOcupado : BOOL; 
END_VAR
VAR
	rtCria : R_TRIG;
	ftCria : F_trig;
	xCria : BOOL;
	fbPLCDBCreate	: FB_PLCDBCreateEvt(sNetID := '', tTimeout := T#30S);

		ColumnInfo : ARRAY[0..3] OF ST_ColumnInfo := [(sName := 'ID', eType := E_ColumnType.BigInt, nLength := 8, sProperty := 'IDENTITY(1,1)'),
												(sName := 'Nome', eType := E_ColumnType.NVarChar, nLength := 80),
												(sName := 'Motores', eType := E_ColumnType.NVarChar, nLength := 255),
												(
				sName := 'Timestamp',
					eType := E_ColumnType.DateTime,
					nLength := 4,
					sProperty := 'DEFAULT CURRENT_TIMESTAMP ON UPDATE CURRENT_TIMESTAMP')];

	i				: INT;
	xGeraMoto		: BOOL;
	diParteBaixa	: DINT;
	diParteAlta		: DINT;

	//Grava valores
	xGravando		: BOOL;
	rtEscrita		: R_TRIG;
	xEscreve		: BOOL;
	EstruturaBanco	: ST_BancoGrupo;
	xEscreveAux		: BOOL;
	sAux			: ARRAY[1..50] OF STRING(80);
	fbPLCDBWrite	: FB_PLCDBWriteEvt(sNetID := '', tTimeout := T#30S); //Bloco para gravar no banco de dados

	ColumnNamesGrava : ARRAY[0..3] OF STRING(50) := ['ID',
													'Nome',
													'Motores',
													'Timestamp'];
	
	/// INICIA
	iEstadoInica : INT;
	
	//Estado 1
	fbPLCDBRead		: FB_PLCDBReadEvt(sNetID := '', tTimeout := T#30S); //Bloco para leitura do banco de dados sem filtro
	iPrimeiraGrupo : INT;
	VetorEstruturaBanco	: ARRAY[0..999] OF ST_BancoGrupo;
	iUltimoGrupo : INT;
	ColumnNamesLe 	: ARRAY[0..3] OF STRING(50) := ['ID',
													'Nome',
													'Motores',
													'Timestamp'];
													
													
													
END_VAR


IF xLicensaValida651641iih THEN
	GeraTabela();
	GeraOsGrupos();
	MaquinaInica();
ELSE	
	ValidaLicensa();
END_IF

ACTION GeraOsGrupos:

diParteBaixa	:= 1;
diParteAlta		:= 100;

IF xGeraMoto THEN

	xEscreve := TRUE;
	rtEscrita(CLK := xEscreve, Q =>);

	IF rtEscrita.q THEN
		xEscreveAux					:= TRUE;
		EstruturaBanco.ID			:= DINT_TO_DWORD(diParteBaixa + i);
		EstruturaBanco.Nome			:= CONCAT('Grupo ', TO_STRING(diParteBaixa + i));
	END_IF

	IF xEscreveAux THEN
		IF fbPLCDBWrite.WriteStruct
			(
				hDBID := INT_TO_UDINT(iNumeroDataBase),
					sTableName := sNomeTabela,
					pRecord := ADR(EstruturaBanco),
					cbRecord := SIZEOF(EstruturaBanco),
					pColumnNames := ADR(ColumnNamesGrava),
					cbColumnNames := SIZEOF(ColumnNamesGrava))
		THEN
			xEscreve := FALSE;
			rtEscrita(CLK := xEscreve, Q =>);
			xEscreveAux	:= FALSE;
			i			:= i + 1;

			IF i > diParteAlta THEN
				xGeraMoto	:= FALSE;
				xOcupado	:= FALSE;
			END_IF
		END_IF
	END_IF

END_IF
END_ACTION

ACTION GeraTabela:

rtCria(CLK := xCriaTabela, Q =>);

IF rtCria.q THEN
	xCria := TRUE;
	xOcupado := TRUE;
END_IF

IF xCria THEN
	IF fbPLCDBCreate.Table(
			hDBID := INT_TO_UDINT(iNumeroDataBase),
			sTableName := sNomeTabela,
			pTableCfg := ADR(ColumnInfo),
			cbTableCfg := SIZEOF(ColumnInfo))
	THEN
		xCria := FALSE;
		xCriaTabela := FALSE;
		xGeraMoto := true;
	END_IF

END_IF
END_ACTION

ACTION MaquinaInica:



CASE iEstadoInica OF
	0: // Esperando começar
		IF xInicia THEN
			iEstadoInica := 1;
		END_IF
		
	1: // Le tudo do banco
	
		iPrimeiraGrupo := DINT_TO_INT(LOWER_BOUND(fbGrupos,1));
		iultimoGrupo := DINT_TO_INT(UPPER_BOUND(fbGrupos,1));
		IF fbPLCDBRead.ReadStruct(
								hDBID:=1 , 
								sTableName:= sNomeTabela, 
								pColumnNames:= ADR(ColumnNamesLe), 
								cbColumnNames:= SIZEOF(ColumnNamesLe), 
								sOrderByColumn:= ColumnNamesLe[0], 
								eOrderType:= E_OrderType.ASC, 
								nStartIndex:= iPrimeiraGrupo, 
								nRecordCount:= iultimoGrupo - iPrimeiraGrupo, 
								pData:= ADR(VetorEstruturaBanco), 
								cbData:= SIZEOF(VetorEstruturaBanco))
		THEN
			iEstadoInica := 0;
			FOR i := iPrimeiraGrupo+1 TO iultimoGrupo DO
				//Faz como se fosse o bloco dele fazendo isso
				fbGrupos[I].EstruturaBanco := VetorEstruturaBanco[i-1];
				//Joga pra onde ele calcula o role
				fbGrupos[I].iEstado := 1;
				//Se for erro ele usa o que ja ta nas persistent
				fbGrupos[I].xAtualizaExternoErro := fbPLCDBRead.bError;
			END_FOR
			xInicia := false;
		END_IF
	
	
	
END_CASE
END_ACTION

END_FUNCTION_BLOCK

// FBs/IHM/FB_GeraListaInterlocksIHM
{attribute 'hide_all_locals'}
FUNCTION_BLOCK FB_GeraListaInterlocksIHM
VAR_IN_OUT
	sListaIHM	: ARRAY[*] OF STRING;
	stMotor		: ARRAY[*] OF st_Partida;
	stSensores	: ARRAY[*] OF st_SensorDigital;
	stOe		: ARRAY[*] OF st_SensorDigital;
	stOs		: ARRAY[*] OF st_SensorDigital;
	stOutros	: ARRAY[*] OF st_OutrosInterlocks;
END_VAR
VAR_INPUT
	xAtualiza : BOOL;
END_VAR
VAR_OUTPUT
	xErro : BOOL;
END_VAR
VAR
	diIHMCima		: DINT;
	diIHMBaixo		: DINT;
	diMotorCima		: DINT;
	diMotorBaixo	: DINT;
	diSensorCima	: DINT;
	diSensorBaixo	: DINT;
	diOutrosCima	: DINT;
	diOutrosBaixo	: DINT;
	i				: DINT;
	iIndex_sLista	: DINT;
	diOeCima		: DINT;
	diOeBaixo		: DINT;
	diOsCima		: DINT;
	diOsBaixo		: DINT;
END_VAR


IF xLicensaValida651641iih THEN
		
	IF xAtualiza THEN
	
		diIHMCima		:= UPPER_BOUND(sListaIHM, 1);
		diIHMBaixo		:= LOWER_BOUND(sListaIHM, 1);
		diMotorCima		:= UPPER_BOUND(stMotor, 1);
		diMotorBaixo	:= LOWER_BOUND(stMotor, 1);
		diSensorCima	:= UPPER_BOUND(stSensores, 1);
		diSensorBaixo	:= LOWER_BOUND(stSensores, 1);
		diOeCima		:= UPPER_BOUND(stOe, 1);
		diOeBaixo		:= LOWER_BOUND(stOe, 1);
		diOsCima		:= UPPER_BOUND(stOs, 1);
		diOsBaixo		:= LOWER_BOUND(stOs, 1);
		diOutrosCima	:= UPPER_BOUND(stOutros, 1);
		diOutrosBaixo	:= LOWER_BOUND(stOutros, 1);
	
		xErro := (diIHMCima - diIHMBaixo) < ((diMotorCima - diMotorBaixo) + (diSensorCima - diSensorBaixo) + (diOutrosCima - diOutrosBaixo) + (diOeCima - diOeBaixo) + (diOsCima - diOsBaixo));
	
		IF xErro THEN
			xAtualiza := FALSE;
		ELSE
			iIndex_sLista := diIHMBaixo;
	
			FOR i := diMotorBaixo TO diMotorCima DO
				IF stMotor[i].BancoDeDados.Tag <> '' THEN
					sListaIHM[iIndex_sLista]	:= stMotor[i].BancoDeDados.Tag;
					iIndex_sLista				:= iIndex_sLista + 1;
				END_IF
			END_FOR
	
			FOR i := diSensorBaixo TO diSensorCima DO
				IF stSensores[i].Banco.Tag <> '' THEN
					sListaIHM[iIndex_sLista]	:= stSensores[i].Banco.Tag;
					iIndex_sLista				:= iIndex_sLista + 1;
				END_IF
			END_FOR
			
			FOR i := diOeBaixo TO diOeCima DO
				IF stOe[i].Banco.Tag <> '' THEN
					sListaIHM[iIndex_sLista]	:= stOe[i].Banco.Tag;
					iIndex_sLista				:= iIndex_sLista + 1;
				END_IF
			END_FOR
			
			FOR i := diOsBaixo TO diOsCima DO
				IF stOs[i].Banco.Tag <> '' THEN
					sListaIHM[iIndex_sLista]	:= stOs[i].Banco.Tag;
					iIndex_sLista				:= iIndex_sLista + 1;
				END_IF
			END_FOR
	
			FOR i := diOutrosBaixo TO diOutrosCima DO
				IF stOutros[i].sTag <> '' THEN
					sListaIHM[iIndex_sLista]	:= stOutros[i].sTag;
					iIndex_sLista				:= iIndex_sLista + 1;
				END_IF
			END_FOR
	
			xAtualiza := FALSE;
		END_IF
	
	END_IF

END_IF

END_FUNCTION_BLOCK

// FBs/Iluminacao/FB_ConfigDoTelerruptor
FUNCTION_BLOCK FB_ConfigDoTelerruptor
VAR_IN_OUT
	stTelerruptor	: ARRAY[*] OF stTelerruptor;
END_VAR
VAR_INPUT
	xInicia			: BOOL;
	xCriaTabela		: BOOL;
	iNumeroDataBase	: INT		:= 1;
	sNomeDataBase	: STRING	:= 'iluminacaoconfig';
END_VAR
VAR_OUTPUT
	xOcupado	: BOOL;
END_VAR
VAR
	
	//Cria table
	rtCria			: R_TRIG;
	xCria			: BOOL;
	fbPLCDBCreate	: FB_PLCDBCreateEvt(sNetID := '', tTimeout := T#30S);
	ColumnInfo : ARRAY[0..2] OF ST_ColumnInfo := [(sName := 'Telerruptor', eType := E_ColumnType.Integer, nLength := 8, sProperty := 'IDENTITY(1,1)'),
												  (sName := 'Tag', eType := E_ColumnType.NVarChar, nLength := 80, sProperty := 'DEFAULT $'SEMTAG$''),
												  (sName := 'Funcao', eType := E_ColumnType.NVarChar, nLength := 80, sProperty := 'DEFAULT $'NADA$'')];
												  
												  
	//Gera os Telerruptores
	diParteBaixa		: DINT;
	diParteAlta			: DINT;
	i					: INT;
	xGeraTelerruptores	: BOOL;
	xEscreve			: BOOL;
	xEscreveAux			: BOOL;
	rtEscrita			: R_TRIG;	
	EstruturaBanco		: ARRAY[0..999] OF ConfigTelerruptorDB;
	fbPLCDBWrite		: FB_PLCDBWriteEvt(sNetID := '', tTimeout := T#30S); //Bloco para gravar no banco de dados
	ColumnNamesGrava	: ARRAY[0..2] OF STRING(50) := ['Telerruptor',
														'Tag',
														'Funcao'
														];
														
														
	//Le os nomes
	xFirstScan		: BOOL := TRUE;
	xLe				: BOOL;
	sCmd			: STRING(1000);
	sTag1			: STRING;
	TagAProcurar	: STRING(80);
	sMensagemErro1	: STRING;
	iIndexGrava		: INT := 0;
	iAux			: DINT;
	diCima			: DINT;
	diBaixo			: DINT;
	nRecords		: UDINT;
	Anterior		: ARRAY[0..999] OF stTelerruptor;
	stPara			: ST_ExpParameter;
	EstruturaBancoLe: ARRAY[0..999] OF ConfigTelerruptorDB;
	eEstado			: enum_LeituradosNomes := enum_LeituradosNomes.eEsperando;
	fbSQLDatabase	: FB_SQLDatabaseEvt(sNetID := '', tTimeout := T#30S);
	fbPLCDBCmd		: FB_PLCDBCmdEvt(sNetID := '', tTimeout := T#30S);
	
	//Grava Nomes Novos
	xGrava			: BOOL;
	xAberto			: BOOL;
	sCmd2			: STRING(1000);
	sMensagemErro2	: STRING;
	Nome			: STRING;
	Vazio			: STRING := '';
	Tag				: STRING;
	Funcao			: STRING;
	arrStr			: ARRAY[1..10] OF STRING(255);
	eEstadoGrava	: enum_GravaNomes := enum_GravaNomes.eEsperando;
	fbSqlCommand		: FB_SQLCommandEvt(sNetID := '', tTimeout := T#30S);
	fbSQLDatabase2	: FB_SQLDatabaseEvt(sNetID := '', tTimeout := T#30S);

END_VAR


IF xFirstScan THEN
	//xLe := TRUE;
	//xCriaTabela := TRUE;
END_IF

IF xInicia THEN
	xLe := TRUE;
	eEstado := enum_LeituradosNomes.eEsperando;
END_IF

GeraTabela();
GeraOsTelerruptores();
LeNomes();
GravaValores();


xFirstScan	:= FALSE;
xInicia		:= FALSE;

ACTION GeraOsTelerruptores:

diParteBaixa	:= LOWER_BOUND(stTelerruptor, 1);
diParteAlta		:= UPPER_BOUND(stTelerruptor, 1);

IF xGeraTelerruptores THEN

	xEscreve := TRUE;
	rtEscrita(CLK := xEscreve, Q =>);

	IF rtEscrita.q THEN
		xEscreveAux						:= TRUE;
		xOcupado						:= TRUE;
		i := DINT_TO_INT(diParteBaixa);
	END_IF

	IF xEscreveAux THEN
		EstruturaBanco[i].Tag := CONCAT('IL', INT_TO_STRING(i));
		EstruturaBanco[i].Telerruptor := INT_TO_DINT(i);
		
		IF fbPLCDBWrite.WriteStruct
		(
			hDBID := INT_TO_UDINT(iNumeroDataBase),
				sTableName := sNomeDataBase,
				pRecord := ADR(EstruturaBanco[i]),
				cbRecord := SIZEOF(EstruturaBanco[i]),
				pColumnNames := ADR(ColumnNamesGrava),
				cbColumnNames := SIZEOF(ColumnNamesGrava))
		THEN
			i := i +1;
		ELSE
			IF fbPLCDBWrite.bError THEN
				IF fbPLCDBWrite.ipTcResult.nEventId = 61 THEN
					xCriaTabela := TRUE;
				END_IF
			END_IF
		END_IF
		
		IF i > diParteAlta THEN
			xOcupado	:= FALSE;
			xEscreve 	:= FALSE;
			rtEscrita(CLK := xEscreve, Q =>);
			xEscreveAux	:= FALSE;
			xGeraTelerruptores := FALSE;
			i := DINT_TO_INT(diParteBaixa);
			
			xLe := TRUE;
			eEstado := enum_LeituradosNomes.eEsperando;
		END_IF

	END_IF
END_IF
END_ACTION

ACTION GeraTabela:

rtCria(CLK := xCriaTabela, Q =>);

IF rtCria.q THEN
	xCria		:= TRUE;
	xOcupado	:= TRUE;
END_IF

IF xCria THEN

	IF fbPLCDBCreate.Table
		(
			hDBID := INT_TO_UDINT(iNumeroDataBase),
				sTableName := sNomeDataBase,
				pTableCfg := ADR(ColumnInfo),
				cbTableCfg := SIZEOF(ColumnInfo))
	THEN
		xCria		:= FALSE;
		xCriaTabela	:= FALSE;
		xOcupado	:= FALSE;
		xGeraTelerruptores	:= TRUE;
		i			:= 1;
	END_IF

END_IF
END_ACTION

ACTION GravaValores:
CASE eEstadoGrava OF
		enum_GravaNomes.eEsperando: //Esperando
			IF xGrava THEN
				IF xAberto THEN
					eEstadoGrava := enum_GravaNomes.eCriaComando;
				ELSE
					eEstadoGrava := enum_GravaNomes.eAbreConexao;
				END_IF
				
			END_IF
			
		enum_GravaNomes.eAbreConexao: //abre conexao
			IF fbSQLDatabase2.Connect(INT_TO_UDINT(iNumeroDataBase)) THEN
				IF fbSQLDatabase2.bError THEN
					{error <'Não conseguiu abrir a conexao no banco do bloco FB_IniciaOsBlocosDeConfigDoMotor 1'>}
					IF fbSQLDatabase2.ipTcResult.ipSourceInfo.sName = 'ADSERR_DEVICE_LICENSENOTFOUND' THEN
						// se der isso ele nao fica tentando e gerando uma caralhada de erro pq nao tem a lisença
						eEstadoGrava := enum_GravaNomes.eParado;
					ELSE
						eEstadoGrava := enum_GravaNomes.eAbreConexao;
					END_IF
					
				ELSE
					IF fbSQLDatabase2.bConnected THEN
						eEstadoGrava := enum_GravaNomes.eCriaComando;
						xAberto := TRUE;
					ELSE
						eEstadoGrava := enum_GravaNomes.eFechaConexao;
						xAberto := FALSE;
					END_IF
				END_IF
			END_IF
			
		enum_GravaNomes.eCriaComando:
			IF fbSQLDatabase2.CreateCmd(ADR(fbSqlCommand)) THEN
				IF fbSQLDatabase2.bError THEN
					eEstadoGrava := enum_GravaNomes.eCriaComando;
				ELSE
					eEstadoGrava := enum_GravaNomes.eGravaNomes;
				END_IF
			END_IF
			
		enum_GravaNomes.eGravaNomes:
	
			//UPDATE `geral`.`iluminacaoconfig` SET `Tag` = 'IL' WHERE (`Telerruptor` = '1');
			
			Nome := stTelerruptor[iIndexGrava].Config.sNome_Funcao;
			Tag := CONCAT(CONCAT('IL', TO_STRING(iIndexGrava)), ' - ');
		
			IF FindAndReplace(
						pSrcString:= ADR(Nome), 
						pDeleteString:= ADR(Tag), 
						pInsertString:= ADR(Vazio), 
						pDstString:= ADR(Funcao), 
						nDstSize:= SIZEOF(Funcao)) = 0  THEN
						
				Funcao := '';	
			END_IF
						
			arrStr[1] := 'UPDATE GERAL.';
			arrStr[2] := sNomeDataBase;
			arrStr[3] := ' SET Funcao = "';
			arrStr[4] := Funcao;
			arrStr[5] :='" WHERE (Telerruptor = "';
			arrStr[6] := TO_STRING(iIndexGrava);
			arrStr[7] := '");';
			
			sCmd2 := F_ConcatArray(sArray:= arrStr); 
	
			IF fbSQLCommand.Execute(pSQLCmd := ADR(sCmd2), cbSQLCmd := SIZEOF(sCmd2))
			THEN
				IF fbSQLCommand.bError THEN
					IF fbSQLCommand.ipTcResult.nEventId = 61 THEN
					// Esse erro acontece quando o database não tá criado, nesse caso ele tenta criar
						eEstadoGrava := enum_GravaNomes.eEsperando;
						xCriaTabela := TRUE;
					ELSE
						eEstadoGrava := enum_GravaNomes.eAbreConexao;
					END_IF
					sMensagemErro2 := 'Nao conseguiu a tag';
				ELSE
					sMensagemErro2	:= 'Conseguiu a tag';
				END_IF
				eEstadoGrava := enum_GravaNomes.eFechaConexao;
				iIndexGrava := 0;
			END_IF
			
		enum_GravaNomes.eFechaConexao:
			IF fbSQLDatabase2.Disconnect() THEN
		
				xGrava := FALSE;
				xLe := TRUE;
		
				IF fbSQLDatabase2.bError THEN
					eEstadoGrava := enum_GravaNomes.eEsperando;
				ELSE
					eEstadoGrava := enum_GravaNomes.eEsperando;
					xAberto := FALSE;
				END_IF
			END_IF

END_CASE
END_ACTION

ACTION LeNomes:

CASE eEstado OF
		enum_LeituradosNomes.eEsperando: //Esperando
			IF xLe THEN
				eEstado := enum_LeituradosNomes.eAbreConexao;
			END_IF
			
		
		enum_LeituradosNomes.eAbreConexao: //abre conexao
			IF fbSqlDatabase.Connect(int_to_udint(iNumeroDataBase)) THEN
				IF fbSqlDatabase.bError THEN
					IF fbSqlDatabase.ipTcResult.ipSourceInfo.sName = 'ADSERR_DEVICE_LICENSENOTFOUND' THEN
						// se der isso ele nao fica tentando e gerando uma caralhada de erro pq nao tem a lisença
						eEstado := enum_LeituradosNomes.eParado;
					ELSE
						eEstado := enum_LeituradosNomes.eAbreConexao;
					END_IF
					
				ELSE
					IF fbSqlDatabase.bConnected THEN
						eEstado := enum_LeituradosNomes.eLeOsNomes;
					END_IF
				END_IF
			END_IF
			
			enum_LeituradosNomes.eLeOsNomes: // le o role
				TagAProcurar		:= sTag1;
				stPara.eParaType	:= E_ExpParameterType.STRING_;
				stPara.nParaSize	:= SIZEOF(TagAProcurar);
				stPara.sParaName	:= 'Tag';
		
				diBaixo	:= LOWER_BOUND(stTelerruptor, 1);
				diCima		:= UPPER_BOUND(stTelerruptor, 1);
		
				// set command with placeholder
				sCmd := CONCAT(CONCAT('SELECT * FROM geral.', sNomeDataBase), ';');
		
				// call functionblock
				IF fbPLCDBCmd.ExecuteDataReturn
					(
						hDBID := INT_TO_UDINT(iNumeroDataBase),
							pExpression := ADR(sCmd),
							cbExpression := SIZEOF(sCmd),
							pData := ADR(TagAProcurar),
							cbData := SIZEOF(TagAProcurar),
							pParameter := ADR(stPara),
							cbParameter := SIZEOF(stPara),
							nStartIndex := DINT_TO_UDINT(diBaixo),
							nRecordCount := DINT_TO_UDINT(diCima),
							pReturnData := ADR(EstruturaBancoLe),
							cbReturnData := SIZEOF(EstruturaBancoLe),
							pRecords := ADR(nRecords))
				THEN
					IF fbPLCDBCmd.bError THEN
						sMensagemErro1 := 'Nao conseguiu a tag';
						{error <'Não conseguiu ler o banco no bloco FB_IniciaOsBlocosDeConfigDoTelerruptor'>}
					ELSE
						sMensagemErro1	:= 'Conseguiu a tag';
						eEstado			:= enum_LeituradosNomes.eFechaConexao;
		
						FOR i := TO_INT(diBaixo) TO TO_INT(diCima) DO
							Anterior[i+1].Config.sNome_Funcao := CONCAT(CONCAT(EstruturaBancoLe[i].Tag, ' - '), EstruturaBancoLe[i].Funcao);
							stTelerruptor[i+1].Config.sNome_Funcao := CONCAT(CONCAT(EstruturaBancoLe[i].Tag, ' - '), EstruturaBancoLe[i].Funcao);
						END_FOR
						
					END_IF
				END_IF
			
			enum_LeituradosNomes.eFechaConexao: // FechaConexao conexao
				IF fbSqlDatabase.Disconnect() THEN
		
					xLe := FALSE;
					xInicia := FALSE;
		
					IF fbSqlDatabase.bError THEN
						{error <'Não conseguiu abrir a conexao no banco do bloco FB_IniciaOsBlocosDeConfigDoMotor 3'>}
						eEstado := enum_LeituradosNomes.eFechaConexao;
					ELSE
						eEstado := enum_LeituradosNomes.eMonitoraTrocaDeNomes;
					END_IF
				END_IF	

			enum_LeituradosNomes.eMonitoraTrocaDeNomes:
				FOR i := TO_INT(diBaixo) TO TO_INT(diCima) DO
					IF (stTelerruptor[i].Config.sNome_Funcao <> Anterior[i].Config.sNome_Funcao) THEN
						Anterior[i].Config.sNome_Funcao := stTelerruptor[i].Config.sNome_Funcao;
						iIndexGrava := i;
						xGrava := TRUE;
					END_IF
				END_FOR						
END_CASE
END_ACTION

END_FUNCTION_BLOCK

// FBs/Partidas/FB_IniciaOsBlocosDeConfigDoMotor
//{attribute 'hide_all_locals'}
FUNCTION_BLOCK FB_IniciaOsBlocosDeConfigDoMotor
VAR_IN_OUT
	fbBlocoConfig	: ARRAY[*] OF FB_ConfigPartidaNoBanco;
	stMotor			: ARRAY[*] OF st_Partida;
	stSensores		: ARRAY[*] OF st_SensorDigital;
	stOe			: ARRAY[*] OF st_SensorDigital;
	stOs			: ARRAY[*] OF st_SensorDigital;
	stOutros		: ARRAY[*] OF st_OutrosInterlocks;
	stEmergencias 	: ARRAY[*] OF st_Emergencia;
END_VAR
VAR_INPUT
	xInicia			: BOOL;
	iNumeroDataBase	: INT		:= 1;
	sNomeDataBase	: STRING	:= 'motoresconfig';
END_VAR
VAR_OUTPUT
END_VAR
VAR
	fbPLCDBCmd			: FB_PLCDBCmdEvt(sNetID := '', tTimeout := T#30S);
	fbSQLDatabase		: FB_SQLDatabaseEvt(sNetID := '', tTimeout := T#30S);
	sCmd				: STRING(1000);
	sCmdUpdate			: STRING(1000);
	stPara				: ST_ExpParameter;
	TagAProcurar		: STRING(80);
	iVoltaDoComando		: T_ULARGE_INTEGER;
	nRecords			: UDINT;
	xProcuraNaTabela	: BOOL;
	EstruturaBanco		: ARRAY[0..999] OF ST_ConfigMotorDB;
	xJogaNoInterlock	: BOOL;
	sTag1				: STRING;
	sTag2				: STRING;
	xEMotor				: BOOL;
	sMensagemErro1		: STRING;
	diCimaMotor			: DINT;
	diBaixoMotor		: DINT;

	iEstado	: INT := 1;
	i		: INT;

	iAux : INT;

	Verdadeiro	: BOOL	:= TRUE;
	Falso		: BOOL	:= FALSE;
	
	sTags : ARRAY[1..4,1..2] OF STRING;
	sEmergencias : ARRAY[1..4] OF STRING;

END_VAR


IF xLicensaValida651641iih THEN

	CASE iEstado OF
		1: //Esperando
			IF xInicia THEN
				iEstado := 2;
			END_IF
	
		2: //abre conexao
			IF fbSqlDatabase.Connect(int_to_udint(iNumeroDataBase)) THEN
				IF fbSqlDatabase.bError THEN
					{error <'Não conseguiu abrir a conexao no banco do bloco FB_IniciaOsBlocosDeConfigDoMotor 1'>}
					IF fbSqlDatabase.ipTcResult.ipSourceInfo.sName = 'ADSERR_DEVICE_LICENSENOTFOUND' THEN
						// se der isso ele nao fica tentando e gerando uma caralhada de erro pq nao tem a lisença
						iEstado := 0;
					ELSE
						iEstado := 2;
					END_IF
					
				ELSE
					IF fbSqlDatabase.bConnected THEN
						iEstado := 3;
					END_IF
				END_IF
			END_IF
	
		3: // le o role
			TagAProcurar		:= sTag1;
			stPara.eParaType	:= E_ExpParameterType.STRING_;
			stPara.nParaSize	:= SIZEOF(TagAProcurar);
			stPara.sParaName	:= 'Tag';
	
			diBaixoMotor	:= LOWER_BOUND(fbBlocoConfig, 1);
			diCimaMotor		:= UPPER_BOUND(fbBlocoConfig, 1);
	
			// set command with placeholder
			//sCmd := 'SELECT * FROM geral.motoresconfig;';
			sCmd := CONCAT(CONCAT('SELECT * FROM geral.', sNomeDataBase), ';');
	
			// call functionblock
			IF fbPLCDBCmd.ExecuteDataReturn
				(
					hDBID := INT_TO_UDINT(iNumeroDataBase),
						pExpression := ADR(sCmd),
						cbExpression := SIZEOF(sCmd),
						pData := ADR(TagAProcurar),
						cbData := SIZEOF(TagAProcurar),
						pParameter := ADR(stPara),
						cbParameter := SIZEOF(stPara),
						nStartIndex := DINT_TO_UDINT(diBaixoMotor - 1),
						nRecordCount := DINT_TO_UDINT(diCimaMotor),
						pReturnData := ADR(EstruturaBanco),
						cbReturnData := SIZEOF(EstruturaBanco),
						pRecords := ADR(nRecords))
			THEN
				IF fbPLCDBCmd.bError THEN
					sMensagemErro1 := 'Nao conseguiu a tag';
					{error <'Não conseguiu ler o banco no bloco FB_IniciaOsBlocosDeConfigDoMotor 2'>}
				ELSE
					sMensagemErro1	:= 'Conseguiu a tag';
					iEstado			:= 4;
	
					FOR i := TO_INT(diBaixoMotor) TO TO_INT(diCimaMotor) DO
						iAux									:= fbBlocoConfig[i].iIndexMotor;
						stMotor[iAux].BancoDeDados				:= EstruturaBanco[i - 1];
						fbBlocoConfig[i].EstadoAtual			:= enum_MaquinaConfigPartidaDB.ExecutaInterlocks;
						fbBlocoConfig[i].xAtualizadoExternamente:= TRUE;
					END_FOR
				END_IF
			END_IF
	
		4:
			FOR i := TO_INT(diBaixoMotor) TO TO_INT(diCimaMotor) DO
				sTags[1,1] := stMotor[i].BancoDeDados.IT1A;
				sTags[1,2] := stMotor[i].BancoDeDados.IT1B;
				sTags[2,1] := stMotor[i].BancoDeDados.IT2A;
				sTags[2,2] := stMotor[i].BancoDeDados.IT2B;
				sTags[3,1] := stMotor[i].BancoDeDados.IT3A;
				sTags[3,2] := stMotor[i].BancoDeDados.IT3B;
				sTags[4,1] := stMotor[i].BancoDeDados.IT4A;
				sTags[4,2] := stMotor[i].BancoDeDados.IT4B;
				
				sEmergencias[1] := stMotor[i].BancoDeDados.Emerg1;			
				sEmergencias[2] := stMotor[i].BancoDeDados.Emerg2;			
				sEmergencias[3] := stMotor[i].BancoDeDados.Emerg3;			
				sEmergencias[4] := stMotor[i].BancoDeDados.Emerg4;
				
				AtualizaTagInterlocks(i,sTags);
				AtualizaTagEmergencias(i,sEmergencias);
			END_FOR
	
			iEstado := 5;
	
		5: // FechaConexao conexao
			IF fbSqlDatabase.Disconnect() THEN
	
				xInicia := FALSE;
	
				IF fbSqlDatabase.bError THEN
					{error <'Não conseguiu abrir a conexao no banco do bloco FB_IniciaOsBlocosDeConfigDoMotor 3'>}
					iEstado := 5;
				ELSE
					iEstado := 1;
				END_IF
			END_IF
	END_CASE

END_IF

METHOD PRIVATE AtualizaTagEmergencias : BOOL
VAR_INPUT
	iInterno : INT;
	sEmergencias : ARRAY[1..4] OF STRING;
END_VAR
VAR
	i : INT;
	iTagI : INT;
END_VAR

FOR iTagI := 1 TO 4 DO
	FOR i := DINT_TO_INT(LOWER_BOUND(stEmergencias, 1)) TO DINT_TO_INT(UPPER_BOUND(stEmergencias, 1)) DO
		IF stEmergencias[i].Banco.Tag = sEmergencias[iTagI] AND sEmergencias[iTagI] <> '' THEN
			EXIT;
		END_IF
	END_FOR
	
	CASE iTagI OF
		1:
			IF i < DINT_TO_INT(UPPER_BOUND(stEmergencias, 1)) THEN
				fbBlocoConfig[iInterno].RefEmer1 REF= stEmergencias[i].En.xEmergenciaOK;
			ELSE
				fbBlocoConfig[iInterno].RefEmer1 REF= Verdadeiro;
			END_IF
		2:
			IF i < DINT_TO_INT(UPPER_BOUND(stEmergencias, 1)) THEN
				fbBlocoConfig[iInterno].RefEmer2 REF= stEmergencias[i].En.xEmergenciaOK;
			ELSE
				fbBlocoConfig[iInterno].RefEmer2 REF= Verdadeiro;
			END_IF		
		3:
			IF i < DINT_TO_INT(UPPER_BOUND(stEmergencias, 1)) THEN
				fbBlocoConfig[iInterno].RefEmer3 REF= stEmergencias[i].En.xEmergenciaOK;
			ELSE
				fbBlocoConfig[iInterno].RefEmer3 REF= Verdadeiro;
			END_IF
		4:
			IF i < DINT_TO_INT(UPPER_BOUND(stEmergencias, 1)) THEN
				fbBlocoConfig[iInterno].RefEmer4 REF= stEmergencias[i].En.xEmergenciaOK;
			ELSE
				fbBlocoConfig[iInterno].RefEmer4 REF= Verdadeiro;
			END_IF
		
	END_CASE
		
END_FOR
END_METHOD

METHOD PRIVATE AtualizaTagInterlocks : BOOL
VAR_INPUT
	iInterno : INT;
	sTags : ARRAY[1..4,1..2] OF STRING;
END_VAR
VAR
	iTagI : INT := 1;
	iTagJ : INT := 1;
	i : INT;
END_VAR

LinkaOsNaoInterlocks(iInterno);

fbBlocoConfig[iInterno].xAtualizadoExternamente := true;
FOR iTagI := 1 TO 4 DO
	FOR iTagJ := 1 TO 2 DO
		IF sTags[iTagi, iTagJ] <> '' THEN
			IF FIND(STR1 := sTags[iTagI, iTagJ], STR2 := 'M') = 1 THEN
				FOR i := DINT_TO_INT(LOWER_BOUND(stMotor, 1)) TO DINT_TO_INT(UPPER_BOUND(stMotor, 1)) DO
					IF stMotor[i].BancoDeDados.Tag = sTags[iTagI, iTagJ] THEN
						EXIT;
					END_IF
				END_FOR

				CASE iTagI OF
					1:
						IF iTagJ = 1 THEN
							fbBlocoConfig[iInterno].RefIT1A REF= stMotor[i].Sa.xNaoLigaProxMotor;
						ELSE
							fbBlocoConfig[iInterno].RefIT1B REF= stMotor[i].Sa.xNaoLigaProxMotor;
						END_IF

					2:
						IF iTagJ = 1 THEN
							fbBlocoConfig[iInterno].RefIT2A REF= stMotor[i].Sa.xNaoLigaProxMotor;
						ELSE
							fbBlocoConfig[iInterno].RefIT2B REF= stMotor[i].Sa.xNaoLigaProxMotor;
						END_IF

					3:
						IF iTagJ = 1 THEN
							fbBlocoConfig[iInterno].RefIT3A REF= stMotor[i].Sa.xNaoLigaProxMotor;
						ELSE
							fbBlocoConfig[iInterno].RefIT3B REF= stMotor[i].Sa.xNaoLigaProxMotor;
						END_IF

					4:
						IF iTagJ = 1 THEN
							fbBlocoConfig[iInterno].RefIT4A REF= stMotor[i].Sa.xNaoLigaProxMotor;
						ELSE
							fbBlocoConfig[iInterno].RefIT4B REF= stMotor[i].Sa.xNaoLigaProxMotor;
						END_IF
				END_CASE
			ELSE
				IF FIND(STR1 := sTags[iTagI, iTagJ], STR2 := 'S') = 1 THEN
					FOR i := DINT_TO_INT(LOWER_BOUND(stMotor, 1)) TO DINT_TO_INT(UPPER_BOUND(stMotor, 1)) DO
						IF stSensores[i].Banco.Tag = sTags[iTagI, iTagJ] THEN
							EXIT;
						END_IF
					END_FOR

					CASE iTagI OF
						1:
							IF iTagJ = 1 THEN
								fbBlocoConfig[iInterno].RefIT1A REF= stSensores[i].Sa.xObjPresente;
							ELSE
								fbBlocoConfig[iInterno].RefIT1B REF= stSensores[i].Sa.xObjPresente;
							END_IF

						2:
							IF iTagJ = 1 THEN
								fbBlocoConfig[iInterno].RefIT2A REF= stSensores[i].Sa.xObjPresente;
							ELSE
								fbBlocoConfig[iInterno].RefIT2B REF= stSensores[i].Sa.xObjPresente;
							END_IF

						3:
							IF iTagJ = 1 THEN
								fbBlocoConfig[iInterno].RefIT3A REF= stSensores[i].Sa.xObjPresente;
							ELSE
								fbBlocoConfig[iInterno].RefIT3B REF= stSensores[i].Sa.xObjPresente;
							END_IF

						4:
							IF iTagJ = 1 THEN
								fbBlocoConfig[iInterno].RefIT4A REF= stSensores[i].Sa.xObjPresente;
							ELSE
								fbBlocoConfig[iInterno].RefIT4B REF= stSensores[i].Sa.xObjPresente;
							END_IF
					END_CASE
				ELSIF FIND(STR1 := sTags[iTagI, iTagJ], STR2 := 'OE') = 1 THEN
					FOR i := DINT_TO_INT(LOWER_BOUND(stMotor, 1)) TO DINT_TO_INT(UPPER_BOUND(stMotor, 1)) DO
						IF stOe[i].Banco.Tag = sTags[iTagI, iTagJ] THEN
							EXIT;
						END_IF
					END_FOR

					CASE iTagI OF
						1:
							IF iTagJ = 1 THEN
								fbBlocoConfig[iInterno].RefIT1A REF= stOe[i].Sa.xObjPresente;
							ELSE
								fbBlocoConfig[iInterno].RefIT1B REF= stOe[i].Sa.xObjPresente;
							END_IF

						2:
							IF iTagJ = 1 THEN
								fbBlocoConfig[iInterno].RefIT2A REF= stOe[i].Sa.xObjPresente;
							ELSE
								fbBlocoConfig[iInterno].RefIT2B REF= stOe[i].Sa.xObjPresente;
							END_IF

						3:
							IF iTagJ = 1 THEN
								fbBlocoConfig[iInterno].RefIT3A REF= stOe[i].Sa.xObjPresente;
							ELSE
								fbBlocoConfig[iInterno].RefIT3B REF= stOe[i].Sa.xObjPresente;
							END_IF

						4:
							IF iTagJ = 1 THEN
								fbBlocoConfig[iInterno].RefIT4A REF= stOe[i].Sa.xObjPresente;
							ELSE
								fbBlocoConfig[iInterno].RefIT4B REF= stOe[i].Sa.xObjPresente;
							END_IF
					END_CASE
				ELSIF FIND(STR1 := sTags[iTagI, iTagJ], STR2 := 'OS') = 1 THEN
					FOR i := DINT_TO_INT(LOWER_BOUND(stMotor, 1)) TO DINT_TO_INT(UPPER_BOUND(stMotor, 1)) DO
						IF stOs[i].Banco.Tag = sTags[iTagI, iTagJ] THEN
							EXIT;
						END_IF
					END_FOR

					CASE iTagI OF
						1:
							IF iTagJ = 1 THEN
								fbBlocoConfig[iInterno].RefIT1A REF= stOs[i].Sa.xObjPresente;
							ELSE
								fbBlocoConfig[iInterno].RefIT1B REF= stOs[i].Sa.xObjPresente;
							END_IF

						2:
							IF iTagJ = 1 THEN
								fbBlocoConfig[iInterno].RefIT2A REF= stOs[i].Sa.xObjPresente;
							ELSE
								fbBlocoConfig[iInterno].RefIT2B REF= stOs[i].Sa.xObjPresente;
							END_IF

						3:
							IF iTagJ = 1 THEN
								fbBlocoConfig[iInterno].RefIT3A REF= stOs[i].Sa.xObjPresente;
							ELSE
								fbBlocoConfig[iInterno].RefIT3B REF= stOs[i].Sa.xObjPresente;
							END_IF

						4:
							IF iTagJ = 1 THEN
								fbBlocoConfig[iInterno].RefIT4A REF= stOs[i].Sa.xObjPresente;
							ELSE
								fbBlocoConfig[iInterno].RefIT4B REF= stOs[i].Sa.xObjPresente;
							END_IF
					END_CASE
				ELSE
					FOR i := DINT_TO_INT(LOWER_BOUND(stOutros, 1)) TO DINT_TO_INT(UPPER_BOUND(stOutros, 1)) DO
						IF stOutros[i].sTag = sTags[iTagI, iTagJ] THEN
							EXIT;
						END_IF
					END_FOR

					CASE iTagI OF
						1:
							IF iTagJ = 1 THEN
								fbBlocoConfig[iInterno].RefIT1A REF= stOutros[i].xEstado;
							ELSE
								fbBlocoConfig[iInterno].RefIT1B REF= stOutros[i].xEstado;
							END_IF

						2:
							IF iTagJ = 1 THEN
								fbBlocoConfig[iInterno].RefIT2A REF= stOutros[i].xEstado;
							ELSE
								fbBlocoConfig[iInterno].RefIT2B REF= stOutros[i].xEstado;
							END_IF

						3:
							IF iTagJ = 1 THEN
								fbBlocoConfig[iInterno].RefIT3A REF= stOutros[i].xEstado;
							ELSE
								fbBlocoConfig[iInterno].RefIT3B REF= stOutros[i].xEstado;
							END_IF

						4:
							IF iTagJ = 1 THEN
								fbBlocoConfig[iInterno].RefIT4A REF= stOutros[i].xEstado;
							ELSE
								fbBlocoConfig[iInterno].RefIT4B REF= stOutros[i].xEstado;
							END_IF
					END_CASE
				END_IF
			END_IF
		ELSE
			CASE iTagI OF
				1:
					IF iTagJ = 1 THEN
						fbBlocoConfig[iInterno].RefIT1A REF= Falso;
					ELSE
						fbBlocoConfig[iInterno].RefIT1B REF= Falso;
					END_IF

				2:
					IF iTagJ = 1 THEN
						fbBlocoConfig[iInterno].RefIT2A REF= Falso;
					ELSE
						fbBlocoConfig[iInterno].RefIT2B REF= Falso;
					END_IF

				3:
					IF iTagJ = 1 THEN
						fbBlocoConfig[iInterno].RefIT3A REF= Falso;
					ELSE
						fbBlocoConfig[iInterno].RefIT3B REF= Falso;
					END_IF

				4:
					IF iTagJ = 1 THEN
						fbBlocoConfig[iInterno].RefIT4A REF= Falso;
					ELSE
						fbBlocoConfig[iInterno].RefIT4B REF= Falso;
					END_IF
			END_CASE
		END_IF
	END_FOR
END_FOR
END_METHOD

METHOD PRIVATE LinkaOsNaoInterlocks : BOOL
VAR_INPUT
	i: INT;
END_VAR



//Se inverte
IF stMotor[i].BancoDeDados.InvIT1A = 1 THEN
	fbBlocoConfig[i].RefInvIT1A REF= Verdadeiro;
ELSE
	fbBlocoConfig[i].RefInvIT1A REF= FALSO;
END_IF

//Operação feita
IF stMotor[i].BancoDeDados.OPIT1 = 1 THEN
	fbBlocoConfig[i].RefOPIT1 REF= Verdadeiro;
ELSE
	fbBlocoConfig[i].RefOPIT1 REF= FALSO;
END_IF

//Se inverte o 1B
IF stMotor[i].BancoDeDados.InvIT1B = 1 THEN
	fbBlocoConfig[i].RefInvIT1B REF= Verdadeiro;
ELSE
	fbBlocoConfig[i].RefInvIT1B REF= FALSO;
END_IF

//Se inverte
IF stMotor[i].BancoDeDados.InvIT2A = 1 THEN
	fbBlocoConfig[i].RefInvIT2A REF= Verdadeiro;
ELSE
	fbBlocoConfig[i].RefInvIT2A REF= FALSO;
END_IF

//Operação feita
IF stMotor[i].BancoDeDados.OPIT2 = 1 THEN
	fbBlocoConfig[i].RefOPIT2 REF= Verdadeiro;
ELSE
	fbBlocoConfig[i].RefOPIT2 REF= FALSO;
END_IF

//Se inverte o 2B
IF stMotor[i].BancoDeDados.InvIT2B = 1 THEN
	fbBlocoConfig[i].RefInvIT2B REF= Verdadeiro;
ELSE
	fbBlocoConfig[i].RefInvIT2B REF= FALSO;
END_IF

//Se inverte
IF stMotor[i].BancoDeDados.InvIT3A = 1 THEN
	fbBlocoConfig[i].RefInvIT3A REF= Verdadeiro;
ELSE
	fbBlocoConfig[i].RefInvIT3A REF= FALSO;
END_IF

//Operação feita
IF stMotor[i].BancoDeDados.OPIT3 = 1 THEN
	fbBlocoConfig[i].RefOPIT3 REF= Verdadeiro;
ELSE
	fbBlocoConfig[i].RefOPIT3 REF= FALSO;
END_IF

//Se inverte o 3B
IF stMotor[i].BancoDeDados.InvIT3B = 1 THEN
	fbBlocoConfig[i].RefInvIT3B REF= Verdadeiro;
ELSE
	fbBlocoConfig[i].RefInvIT3B REF= FALSO;
END_IF

//Se inverte
IF stMotor[i].BancoDeDados.InvIT4A = 1 THEN
	fbBlocoConfig[i].RefInvIT4A REF= Verdadeiro;
ELSE
	fbBlocoConfig[i].RefInvIT4A REF= FALSO;
END_IF

//Operação feita
IF stMotor[i].BancoDeDados.OPIT4 = 1 THEN
	fbBlocoConfig[i].RefOPIT4 REF= Verdadeiro;
ELSE
	fbBlocoConfig[i].RefOPIT4 REF= FALSO;
END_IF

//Se inverte o 4B
IF stMotor[i].BancoDeDados.InvIT4B = 1 THEN
	fbBlocoConfig[i].RefInvIT4B REF= Verdadeiro;
ELSE
	fbBlocoConfig[i].RefInvIT4B REF= FALSO;
END_IF
END_METHOD

END_FUNCTION_BLOCK

// FBs/Partidas/FB_ConfigPartidaNoBanco
{attribute 'hide_all_locals'}
FUNCTION_BLOCK FB_ConfigPartidaNoBanco
VAR_IN_OUT
	stMotor			: ARRAY[*] OF st_Partida;
	stSensores		: ARRAY[*] OF st_SensorDigital;
	stOe			: ARRAY[*] OF st_SensorDigital;
	stOs			: ARRAY[*] OF st_SensorDigital;
	stOutros		: ARRAY[*] OF st_OutrosInterlocks;
	stEmergencias 	: ARRAY[*] OF st_Emergencia;
	iAtualizandoAtual : INT;
END_VAR
VAR_INPUT
	// 0 = or 			1 = and

	//xEscreve				: BOOL;
	xLe						: BOOL;
	iNumeroDataBase			: INT		:= 1;
	sNomeDataBase			: STRING	:= 'motoresconfig';
	iIndexMotor				: INT;
	EstadoAtual				: enum_MaquinaConfigPartidaDB;
	xAtualizadoExternamente	: BOOL;
	xNaoAtualiza			: BOOL;
	iMaxAtualizando			: INT := 50;
	
	RefEmer1	: REFERENCE TO BOOL; 	
	RefEmer2	: REFERENCE TO BOOL; 	
	RefEmer3	: REFERENCE TO BOOL; 	
	RefEmer4	: REFERENCE TO BOOL; 

	RefInvIT1A	: REFERENCE TO BOOL;
	RefIT1A		: REFERENCE TO BOOL;
	RefOPIT1	: REFERENCE TO BOOL;
	RefInvIT1B	: REFERENCE TO BOOL;
	RefIT1B		: REFERENCE TO BOOL;

	RefInvIT2A	: REFERENCE TO BOOL;
	RefIT2A		: REFERENCE TO BOOL;
	RefOPIT2	: REFERENCE TO BOOL;
	RefInvIT2B	: REFERENCE TO BOOL;
	RefIT2B		: REFERENCE TO BOOL;

	RefInvIT3A	: REFERENCE TO BOOL;
	RefIT3A		: REFERENCE TO BOOL;
	RefOPIT3	: REFERENCE TO BOOL;
	RefInvIT3B	: REFERENCE TO BOOL;
	RefIT3B		: REFERENCE TO BOOL;

	RefInvIT4A	: REFERENCE TO BOOL;
	RefIT4A		: REFERENCE TO BOOL;
	RefOPIT4	: REFERENCE TO BOOL;
	RefInvIT4B	: REFERENCE TO BOOL;
	RefIT4B		: REFERENCE TO BOOL;
END_VAR
VAR_OUTPUT
	xOcupado	: BOOL;
	xEmergencia	: BOOL;
	xInterlock1	: BOOL;
	xInterlock2	: BOOL;
	xInterlock3	: BOOL;
	xInterlock4	: BOOL;
END_VAR
VAR

	//Interlock
	A	: BOOL;
	B	: BOOL;
	C	: BOOL;

	Verdadeiro	: BOOL	:= TRUE;
	Falso		: BOOL	:= FALSE;

	// geral
	i				: INT;
	iAux			: INT;
	iTag			: INT;
	EstruturaBanco	: ARRAY[0..1] OF Teknike_Partidas.ST_ConfigMotorDB;

	//Comando que pega o Id do motor

	fbPLCDBCmd				: FB_PLCDBCmdEvt(sNetID := '', tTimeout := T#30S);
	sCmd					: STRING(1000);
	sCmdUpdate				: STRING(1000);
	stPara					: ST_ExpParameter;
	TagAProcurar			: STRING(80);
	iVoltaDoComando			: T_ULARGE_INTEGER;
	nRecords				: UDINT;
	xProcuraNaTabela		: BOOL;
	EstruturaBancoInterlock	: Teknike_Partidas.ST_ConfigMotorDB;
	xJogaNoInterlock		: BOOL;
	sTag1					: ARRAY[1..4] OF STRING;
	sTag2					: ARRAY[1..4] OF STRING;
	sEmergencias			: ARRAY[1..4] OF STRING;
	xEMotor					: BOOL;

	//Grava valores
	xGravando			: BOOL;
	EstruturaAnterior	: Teknike_Partidas.ST_ConfigMotorDB;
	rtEscrita			: R_TRIG;
	xEscreveAux			: BOOL;
	sAux				: ARRAY[0..60] OF STRING(80);
	fbSQLDatabase		: FB_SQLDatabaseEvt(sNetID := '', tTimeout := T#30S);
	fbSqlCommand		: FB_SQLCommandEvt(sNetID := '', tTimeout := T#30S);
	fbPLCDBWrite		: FB_PLCDBWriteEvt(sNetID := '', tTimeout := T#30S); //Bloco para gravar no banco de dados

	ColumnNamesGrava : ARRAY[0..26] OF STRING(50) := ['Motor',
														'Tag',
														'Funcao',

														'InvIT1A',
														'IT1A',
														'OPIT1',
														'InvIT1B',
														'IT1B',

														'InvIT2A',
														'IT2A',
														'OPIT2',
														'InvIT2B',
														'IT2B',

														'InvIT3A',
														'IT3A',
														'OPIT3',
														'InvIT3B',
														'IT3B',

														'InvIT4A',
														'IT4A',
														'OPIT4',
														'InvIT4B',
														'IT4B',

														'Emerg1',
														'Emerg2',
														'Emerg3',
														'Emerg4'];

	//Ler valores
	rtAtualiza		: R_TRIG;
	xAtualiza		: BOOL;
	fbPLCDBRead		: FB_PLCDBReadEvt(sNetID := '', tTimeout := T#30S); //Bloco para leitura do banco de dados sem filtro
	sMensagemErro1	: STRING;

	ColumnNames : ARRAY[0..27] OF STRING(50) := ['Motor',
												'Tag',
												'Funcao',

												'InvIT1A',
												'IT1A',
												'OPIT1',
												'InvIT1B',
												'IT1B',

												'InvIT2A',
												'IT2A',
												'OPIT2',
												'InvIT2B',
												'IT2B',

												'InvIT3A',
												'IT3A',
												'OPIT3',
												'InvIT3B',
												'IT3B',

												'InvIT4A',
												'IT4A',
												'OPIT4',
												'InvIT4B',
												'IT4B',

												'Emerg1',
												'Emerg2',
												'Emerg3',
												'Emerg4',

												'Timestamp'];

	xFirstScan : BOOL := TRUE;

	tonFirstScan		: ton;
	xAindaNaoIniciou	: BOOL;
	
	xDiferenteDoAnterior : BOOL;
	
	bControleAtualizando : B_TRIG;
	xTemQueAtualizarSQL : BOOL;
END_VAR


IF xLicensaValida651641iih THEN	
	
	xNaoAtualiza := iMaxAtualizando < iAtualizandoAtual AND NOT xOcupado;
	
	TrocaEstadoLeitura();
	ExecutaEstadoLeitura();
	
	
	xInterlock4 := stMotor[iIndexMotor].En.xInterLock_4;
	xInterlock1 := stMotor[iIndexMotor].En.xInterLock_1;
	xInterlock2 := stMotor[iIndexMotor].En.xInterLock_2;
	xInterlock3 := stMotor[iIndexMotor].En.xInterLock_3;
	xEmergencia := stMotor[iIndexMotor].En.xEmergenciaOK;
	
	
	bControleAtualizando(CLK:=xOcupado , Q=> );
	IF bControleAtualizando.q THEN
		IF xOcupado THEN
			iAtualizandoAtual := iAtualizandoAtual + 1;
		ELSE
			iAtualizandoAtual := iAtualizandoAtual - 1;
		END_IF
	END_IF
	
	xFirstScan := FALSE;

END_IF

ACTION CalculaEmergencia:


IF __ISVALIDREF(RefEmer1) AND __ISVALIDREF(RefEmer2) AND __ISVALIDREF(RefEmer3) AND __ISVALIDREF(RefEmer4) THEN
	stMotor[iIndexMotor].En.xEmergenciaOK := RefEmer1 AND RefEmer2 AND RefEmer3 AND RefEmer4;
	
	stMotor[iIndexMotor].LeiturasInversorIHM.xStatusEmergencias[1] := RefEmer1;
	stMotor[iIndexMotor].LeiturasInversorIHM.xStatusEmergencias[2] := RefEmer2;
	stMotor[iIndexMotor].LeiturasInversorIHM.xStatusEmergencias[3] := RefEmer3;
	stMotor[iIndexMotor].LeiturasInversorIHM.xStatusEmergencias[4] := RefEmer4;
END_IF
END_ACTION

ACTION CalculaInterlock:
	// 0 = or 			1 = and
stMotor[iIndexMotor].En.xInterLock_1 := FALSE;

IF LEN(stMotor[iIndexMotor].BancoDeDados.IT1A) > 0 THEN
	IF __ISVALIDREF(RefIT1A) AND __ISVALIDREF(RefInvIT1A) THEN
		stMotor[iIndexMotor].En.xInterLock_1 := RefInvIT1A XOR RefIT1A;
		
		IF LEN(stMotor[iIndexMotor].BancoDeDados.IT1B) > 0 THEN
			IF __ISVALIDREF(RefIT1B) AND __ISVALIDREF(RefInvIT1B) AND __ISVALIDREF(RefOPIT1) AND __ISVALIDREF(RefInvIT1B) THEN
				A	:= (RefInvIT1A XOR RefIT1A);
				B	:=  RefOPIT1;
				C	:= (RefInvIT1B XOR RefIT1B);
				//Gerado pelo mapa de Karnaugh
				stMotor[iIndexMotor].En.xInterLock_1 := (A AND C) OR (NOT B AND C) OR (A AND NOT B);
				stMotor[iIndexMotor].LeiturasInversorIHM.xStatusInterlocks[1,1] := A;
				stMotor[iIndexMotor].LeiturasInversorIHM.xStatusInterlocks[1,2] := B;
			END_IF
		END_IF
	END_IF
ELSE
	stMotor[iIndexMotor].En.xInterLock_1 := FALSE;
	stMotor[iIndexMotor].LeiturasInversorIHM.xStatusInterlocks[1,1] := FALSE;
	stMotor[iIndexMotor].LeiturasInversorIHM.xStatusInterlocks[1,2] := FALSE;
END_IF



stMotor[iIndexMotor].En.xInterLock_2 := FALSE;

IF LEN(stMotor[iIndexMotor].BancoDeDados.IT2A) > 0 THEN
	IF __ISVALIDREF(RefIT2A) AND __ISVALIDREF(RefInvIT2A) THEN
		stMotor[iIndexMotor].En.xInterLock_2 := RefInvIT2A XOR RefIT2A;
	
		IF LEN(stMotor[iIndexMotor].BancoDeDados.IT2B) > 0 THEN
			IF __ISVALIDREF(RefIT2B) AND __ISVALIDREF(RefInvIT2B) AND __ISVALIDREF(RefOPIT2) AND __ISVALIDREF(RefInvIT2B) THEN
				A	:= (RefInvIT2A XOR RefIT2A);
				B	:= RefOPIT2;
				C	:= (RefInvIT2B XOR RefIT2B);
				//Gerado pelo mapa de Karnaugh
				stMotor[iIndexMotor].En.xInterLock_2 := (A AND C) OR (NOT B AND C) OR (A AND NOT B);
				stMotor[iIndexMotor].LeiturasInversorIHM.xStatusInterlocks[2,1] := A;
				stMotor[iIndexMotor].LeiturasInversorIHM.xStatusInterlocks[2,2] := B;
			END_IF
		END_IF
	END_IF
ELSE
	stMotor[iIndexMotor].En.xInterLock_2 := FALSE;
	stMotor[iIndexMotor].LeiturasInversorIHM.xStatusInterlocks[2,1] := FALSE;
	stMotor[iIndexMotor].LeiturasInversorIHM.xStatusInterlocks[2,2] := FALSE;
END_IF




stMotor[iIndexMotor].En.xInterLock_3 := FALSE;

IF LEN(stMotor[iIndexMotor].BancoDeDados.IT3A) > 0 THEN
	IF __ISVALIDREF(RefIT3A) AND __ISVALIDREF(RefInvIT3A) THEN
		stMotor[iIndexMotor].En.xInterLock_3 := RefInvIT3A XOR RefIT3A;
	
		IF LEN(stMotor[iIndexMotor].BancoDeDados.IT3B) > 0 THEN
			IF __ISVALIDREF(RefIT3B) AND __ISVALIDREF(RefInvIT3B) AND __ISVALIDREF(RefOPIT3) AND __ISVALIDREF(RefInvIT3B) THEN
				A	:= (RefInvIT3A XOR RefIT3A);
				B	:= RefOPIT3;
				C	:= (RefInvIT3B XOR RefIT3B);
				//Gerado pelo mapa de Karnaugh
				stMotor[iIndexMotor].En.xInterLock_3 := (A AND C) OR (NOT B AND C) OR (A AND NOT B);
				stMotor[iIndexMotor].LeiturasInversorIHM.xStatusInterlocks[3,1] := A;
				stMotor[iIndexMotor].LeiturasInversorIHM.xStatusInterlocks[3,2] := B;
			END_IF
		END_IF
	END_IF
ELSE
	stMotor[iIndexMotor].En.xInterLock_3 := FALSE;
	stMotor[iIndexMotor].LeiturasInversorIHM.xStatusInterlocks[3,1] := FALSE;
	stMotor[iIndexMotor].LeiturasInversorIHM.xStatusInterlocks[3,2] := FALSE;
END_IF





stMotor[iIndexMotor].En.xInterLock_4 := FALSE;

IF LEN(stMotor[iIndexMotor].BancoDeDados.IT4A) > 0 THEN
	IF __ISVALIDREF(RefIT4A) AND __ISVALIDREF(RefInvIT4A) THEN
		stMotor[iIndexMotor].En.xInterLock_4 := RefInvIT4A XOR RefIT4A;
	
		IF LEN(stMotor[iIndexMotor].BancoDeDados.IT4B) > 0 THEN
			IF __ISVALIDREF(RefIT4B) AND __ISVALIDREF(RefInvIT4B) AND __ISVALIDREF(RefOPIT4) AND __ISVALIDREF(RefInvIT4B) THEN
				A	:= (RefInvIT4A XOR RefIT4A);
				B	:= RefOPIT4;
				C	:= (RefInvIT4B XOR RefIT4B);
				//Gerado pelo mapa de Karnaugh
				stMotor[iIndexMotor].En.xInterLock_4 := (A AND C) OR (NOT B AND C) OR (A AND NOT B);
				stMotor[iIndexMotor].LeiturasInversorIHM.xStatusInterlocks[4,1] := A;
				stMotor[iIndexMotor].LeiturasInversorIHM.xStatusInterlocks[4,2] := B;
			END_IF
		END_IF
	END_IF
ELSE
	stMotor[iIndexMotor].En.xInterLock_4 := FALSE;
	stMotor[iIndexMotor].LeiturasInversorIHM.xStatusInterlocks[4,1] := FALSE;
	stMotor[iIndexMotor].LeiturasInversorIHM.xStatusInterlocks[4,2] := FALSE;
END_IF
END_ACTION

ACTION ExecutaEstadoLeitura:

CASE EstadoAtual OF

	enum_MaquinaConfigPartidaDB.Esperando:
		xLe := xLe;

	enum_MaquinaConfigPartidaDB.AbreConexao:
		iAux := iAux;

	enum_MaquinaConfigPartidaDB.CriaComando:
		iAux := iAux;

	enum_MaquinaConfigPartidaDB.Gravando:
		sAux[0] := CONCAT(CONCAT('UPDATE geral.',sNomeDataBase),' SET ');

		IF stMotor[iIndexMotor].BancoDeDados.Tag <> '' THEN
			sAux[1]	:= 'Tag = $'';
			sAux[2]	:= CONCAT((stMotor[iIndexMotor].BancoDeDados.Tag), '$', ');
		ELSE
			sAux[1]	:= '';
			sAux[2]	:= '';
		END_IF

		sAux[3]		:= 'Funcao = $'';
		sAux[4]		:= (stMotor[iIndexMotor].BancoDeDados.Funcao);
		sAux[5]		:= '$', InvIT1A = $'';
		sAux[6]		:= INT_TO_STRING(stMotor[iIndexMotor].BancoDeDados.InvIT1A);
		sAux[7]		:= '$', IT1A = $'';
		sAux[8]		:= (stMotor[iIndexMotor].BancoDeDados.IT1A);
		sAux[9]		:= '$', OPIT1 = $'';
		sAux[10]	:= INT_TO_STRING(stMotor[iIndexMotor].BancoDeDados.OPIT1);
		sAux[11]	:= '$', InvIT1B = $'';
		sAux[12]	:= INT_TO_STRING(stMotor[iIndexMotor].BancoDeDados.InvIT1B);
		sAux[13]	:= '$', IT1B = $'';
		sAux[14]	:= (stMotor[iIndexMotor].BancoDeDados.IT1B);
		sAux[15]	:= '$', InvIT2A = $'';
		sAux[16]	:= INT_TO_STRING(stMotor[iIndexMotor].BancoDeDados.InvIT2A);
		sAux[17]	:= '$', IT2A = $'';
		sAux[18]	:= (stMotor[iIndexMotor].BancoDeDados.IT2A);
		sAux[19]	:= '$', OPIT2 = $'';
		sAux[20]	:= INT_TO_STRING(stMotor[iIndexMotor].BancoDeDados.OPIT2);
		sAux[21]	:= '$', InvIT2B = $'';
		sAux[22]	:= INT_TO_STRING(stMotor[iIndexMotor].BancoDeDados.InvIT2B);
		sAux[23]	:= '$', IT2B = $'';
		sAux[24]	:= (stMotor[iIndexMotor].BancoDeDados.IT2B);
		sAux[25]	:= '$', InvIT3A = $'';
		sAux[26]	:= INT_TO_STRING(stMotor[iIndexMotor].BancoDeDados.InvIT3A);
		sAux[27]	:= '$', IT3A = $'';
		sAux[28]	:= (stMotor[iIndexMotor].BancoDeDados.IT3A);
		sAux[29]	:= '$', OPIT3 = $'';
		sAux[30]	:= INT_TO_STRING(stMotor[iIndexMotor].BancoDeDados.OPIT3);
		sAux[31]	:= '$', InvIT3B = $'';
		sAux[32]	:= INT_TO_STRING(stMotor[iIndexMotor].BancoDeDados.InvIT3B);
		sAux[33]	:= '$', IT3B = $'';
		sAux[34]	:= (stMotor[iIndexMotor].BancoDeDados.IT3B);
		sAux[35]	:= '$', InvIT4A = $'';
		sAux[36]	:= INT_TO_STRING(stMotor[iIndexMotor].BancoDeDados.InvIT4A);
		sAux[37]	:= '$', IT4A = $'';
		sAux[38]	:= (stMotor[iIndexMotor].BancoDeDados.IT4A);
		sAux[39]	:= '$', OPIT4 = $'';
		sAux[40]	:= INT_TO_STRING(stMotor[iIndexMotor].BancoDeDados.OPIT4);
		sAux[41]	:= '$', InvIT4B = $'';
		sAux[42]	:= INT_TO_STRING(stMotor[iIndexMotor].BancoDeDados.InvIT4B);
		sAux[43]	:= '$', IT4B = $'';
		sAux[44]	:= (stMotor[iIndexMotor].BancoDeDados.IT4B);
		
		sAux[45]	:= '$', Emerg1 = $'';
		sAux[46]	:= (stMotor[iIndexMotor].BancoDeDados.Emerg1);		
		sAux[47]	:= '$', Emerg2 = $'';
		sAux[48]	:= (stMotor[iIndexMotor].BancoDeDados.Emerg2);		
		sAux[49]	:= '$', Emerg3 = $'';
		sAux[50]	:= (stMotor[iIndexMotor].BancoDeDados.Emerg3);		
		sAux[51]	:= '$', Emerg4 = $'';
		sAux[52]	:= (stMotor[iIndexMotor].BancoDeDados.Emerg4);
		
		sAux[53]	:= '$' WHERE (Motor = $'';
		sAux[54]	:= INT_TO_STRING(iIndexMotor);
		sAux[55]	:= '$');';
		sCmdUpdate	:= F_ConcatArray1000(sArray := sAux);

	enum_MaquinaConfigPartidaDB.FechaConexao:
		iAux := iAux;

	enum_MaquinaConfigPartidaDB.LendoEleMesmo:
		
		
		IF NOT xNaoAtualiza THEN
			IF fbPLCDBRead.ReadStruct
				(
					hDBID := INT_TO_UDINT(iNumeroDataBase),
						sTableName := sNomeDataBase,
						pColumnNames := ADR(ColumnNames),
						cbColumnNames := SIZEOF(ColumnNames),
						sOrderByColumn := ColumnNames[0],
						eOrderType := E_OrderType.ASC,
						nStartIndex := INT_TO_UDINT(iIndexMotor - 1),
						nRecordCount := 2,
						pData := ADR(EstruturaBanco),
						cbData := SIZEOF(EstruturaBanco))
			THEN
	
				IF fbPLCDBRead.bError THEN
					{error <'Não conseguiu ler ele mesmo no banco no bloco FB_ConfigPartidaNoBanco 4'>}
					sMensagemErro1 := 'Erro ao ler o banco de dados';
				ELSE
					sMensagemErro1								:= 'Leitura dos dados com sucesso';
					sTag1[1]									:= EstruturaBanco[0].IT1A;
					sTag2[1]									:= EstruturaBanco[0].IT1B;
					sTag1[2]									:= EstruturaBanco[0].IT2A;
					sTag2[2]									:= EstruturaBanco[0].IT2B;
					sTag1[3]									:= EstruturaBanco[0].IT3A;
					sTag2[3]									:= EstruturaBanco[0].IT3B;
					sTag1[4]									:= EstruturaBanco[0].IT4A;
					sTag2[4]									:= EstruturaBanco[0].IT4B;
					stMotor[iIndexMotor].BancoDeDados			:= EstruturaBanco[0];
					
					sEmergencias[1] := EstruturaBanco[0].Emerg1;			
					sEmergencias[2] := EstruturaBanco[0].Emerg2;			
					sEmergencias[3] := EstruturaBanco[0].Emerg3;			
					sEmergencias[4] := EstruturaBanco[0].Emerg4;
					
				END_IF
	
				xLe := FALSE;
				ZeraReferencias();
			END_IF
		END_IF

	enum_MaquinaConfigPartidaDB.LinkaOsNaoInterlock:

		LinkaOsNaoInterlock();

	enum_MaquinaConfigPartidaDB.ProcuraTag1:
		IF sTag1[iTag] <> '' THEN	
			CASE iTag OF
				1:
					xDiferenteDoAnterior := sTag1[iTag] <> EstruturaAnterior.IT1A;
	
				2:
					xDiferenteDoAnterior := sTag1[iTag] <> EstruturaAnterior.IT2A;
	
				3:
					xDiferenteDoAnterior := sTag1[iTag] <> EstruturaAnterior.IT3A;
	
				4:
					xDiferenteDoAnterior := sTag1[iTag] <> EstruturaAnterior.IT4A;
			END_CASE 
		
			IF xDiferenteDoAnterior THEN
				IF FIND(STR1 := sTag1[iTag], STR2 := 'M') = 1 THEN
	
					TagAProcurar		:= sTag1[iTag];
					stPara.eParaType	:= E_ExpParameterType.STRING_;
					stPara.nParaSize	:= SIZEOF(TagAProcurar);
					stPara.sParaName	:= 'Tag';
	
					// set command with placeholder
					sCmd := CONCAT(CONCAT(CONCAT(CONCAT('SELECT motor FROM geral.',sNomeDataBase),' where Tag=$''), TagAProcurar), '$';');
	
					// call functionblock
					IF NOT xNaoAtualiza THEN
						IF fbPLCDBCmd.ExecuteDataReturn
							(
								hDBID := 1,
									pExpression := ADR(sCmd),
									cbExpression := SIZEOF(sCmd),
									pData := ADR(TagAProcurar),
									cbData := SIZEOF(TagAProcurar),
									pParameter := ADR(stPara),
									cbParameter := SIZEOF(stPara),
									nStartIndex := 0,
									nRecordCount := 1,
									pReturnData := ADR(iVoltaDoComando),
									cbReturnData := SIZEOF(iVoltaDoComando),
									pRecords := ADR(nRecords))
						THEN
							IF fbPLCDBCmd.bError THEN
								{error <'Não conseguiu ler TAG1A no banco no bloco FB_ConfigPartidaNoBanco 5'>}
								sMensagemErro1 := 'Nao conseguiu a tag';
							ELSE
								sMensagemErro1 := 'Conseguiu a tag';
		
								CASE iTag OF
									1:
										RefIT1A REF= stMotor[iVoltaDoComando.dwLowPart].Sa.xNaoLigaProxMotor;
		
									2:
										RefIT2A REF= stMotor[iVoltaDoComando.dwLowPart].Sa.xNaoLigaProxMotor;
		
									3:
										RefIT3A REF= stMotor[iVoltaDoComando.dwLowPart].Sa.xNaoLigaProxMotor;
		
									4:
										RefIT4A REF= stMotor[iVoltaDoComando.dwLowPart].Sa.xNaoLigaProxMotor;
								END_CASE
		
								iTag := iTag + 1;
							END_IF
						END_IF
					END_IF
				ELSE
					
				
				
				
					IF FIND(STR1 := sTag1[iTag], STR2 := 'S') = 1 THEN
						//quando for sensor
						TagAProcurar		:= sTag1[iTag];
						stPara.eParaType	:= E_ExpParameterType.STRING_;
						stPara.nParaSize	:= SIZEOF(TagAProcurar);
						stPara.sParaName	:= 'Tag';
	
						// set command with placeholder
						sCmd := CONCAT(CONCAT('SELECT sensor FROM geral.sensoresconfig where Tag=$'', TagAProcurar), '$';');
	
						// call functionblock
						IF NOT xNaoAtualiza THEN
							IF fbPLCDBCmd.ExecuteDataReturn
								(
									hDBID := 1,
										pExpression := ADR(sCmd),
										cbExpression := SIZEOF(sCmd),
										pData := ADR(TagAProcurar),
										cbData := SIZEOF(TagAProcurar),
										pParameter := ADR(stPara),
										cbParameter := SIZEOF(stPara),
										nStartIndex := 0,
										nRecordCount := 1,
										pReturnData := ADR(iVoltaDoComando),
										cbReturnData := SIZEOF(iVoltaDoComando),
										pRecords := ADR(nRecords))
							THEN
								IF fbPLCDBCmd.bError THEN
									sMensagemErro1 := 'Nao conseguiu a tag';
									{error <'Não conseguiu ler TAG1B no banco no bloco FB_ConfigPartidaNoBanco 6'>}
								ELSE
									sMensagemErro1 := 'Conseguiu a tag';
		
									CASE iTag OF
										1:
											RefIT1A REF= stSensores[iVoltaDoComando.dwLowPart].Sa.xObjPresente;
		
										2:
											RefIT2A REF= stSensores[iVoltaDoComando.dwLowPart].Sa.xObjPresente;
		
										3:
											RefIT3A REF= stSensores[iVoltaDoComando.dwLowPart].Sa.xObjPresente;
		
										4:
											RefIT4A REF= stSensores[iVoltaDoComando.dwLowPart].Sa.xObjPresente;
									END_CASE
		
									iTag := iTag + 1;
								END_IF
							END_IF
						END_IF
					ELSIF FIND(STR1 := sTag1[iTag], STR2 := 'OE') = 1 THEN
						//quando for sensor
						TagAProcurar		:= sTag1[iTag];
						stPara.eParaType	:= E_ExpParameterType.STRING_;
						stPara.nParaSize	:= SIZEOF(TagAProcurar);
						stPara.sParaName	:= 'Tag';
	
						// set command with placeholder
						sCmd := CONCAT(CONCAT('SELECT sensor FROM geral.Oeconfig where Tag=$'', TagAProcurar), '$';');
	
						// call functionblock
						IF NOT xNaoAtualiza THEN
							IF fbPLCDBCmd.ExecuteDataReturn
								(
									hDBID := 1,
										pExpression := ADR(sCmd),
										cbExpression := SIZEOF(sCmd),
										pData := ADR(TagAProcurar),
										cbData := SIZEOF(TagAProcurar),
										pParameter := ADR(stPara),
										cbParameter := SIZEOF(stPara),
										nStartIndex := 0,
										nRecordCount := 1,
										pReturnData := ADR(iVoltaDoComando),
										cbReturnData := SIZEOF(iVoltaDoComando),
										pRecords := ADR(nRecords))
							THEN
								IF fbPLCDBCmd.bError THEN
									sMensagemErro1 := 'Nao conseguiu a tag';
									{error <'Não conseguiu ler TAG1B no banco no bloco FB_ConfigPartidaNoBanco 6'>}
								ELSE
									sMensagemErro1 := 'Conseguiu a tag';
		
									CASE iTag OF
										1:
											RefIT1A REF= stOe[iVoltaDoComando.dwLowPart].Sa.xObjPresente;
		
										2:
											RefIT2A REF= stOe[iVoltaDoComando.dwLowPart].Sa.xObjPresente;
		
										3:
											RefIT3A REF= stOe[iVoltaDoComando.dwLowPart].Sa.xObjPresente;
		
										4:
											RefIT4A REF= stOe[iVoltaDoComando.dwLowPart].Sa.xObjPresente;
									END_CASE
		
									iTag := iTag + 1;
								END_IF
							END_IF
						END_IF
					ELSIF FIND(STR1 := sTag1[iTag], STR2 := 'OS') = 1 THEN
						//quando for sensor
						TagAProcurar		:= sTag1[iTag];
						stPara.eParaType	:= E_ExpParameterType.STRING_;
						stPara.nParaSize	:= SIZEOF(TagAProcurar);
						stPara.sParaName	:= 'Tag';
	
						// set command with placeholder
						sCmd := CONCAT(CONCAT('SELECT sensor FROM geral.Osconfig where Tag=$'', TagAProcurar), '$';');
	
						// call functionblock
						IF NOT xNaoAtualiza THEN
							IF fbPLCDBCmd.ExecuteDataReturn
								(
									hDBID := 1,
										pExpression := ADR(sCmd),
										cbExpression := SIZEOF(sCmd),
										pData := ADR(TagAProcurar),
										cbData := SIZEOF(TagAProcurar),
										pParameter := ADR(stPara),
										cbParameter := SIZEOF(stPara),
										nStartIndex := 0,
										nRecordCount := 1,
										pReturnData := ADR(iVoltaDoComando),
										cbReturnData := SIZEOF(iVoltaDoComando),
										pRecords := ADR(nRecords))
							THEN
								IF fbPLCDBCmd.bError THEN
									sMensagemErro1 := 'Nao conseguiu a tag';
									{error <'Não conseguiu ler TAG1B no banco no bloco FB_ConfigPartidaNoBanco 6'>}
								ELSE
									sMensagemErro1 := 'Conseguiu a tag';
		
									CASE iTag OF
										1:
											RefIT1A REF= stOs[iVoltaDoComando.dwLowPart].Sa.xObjPresente;
		
										2:
											RefIT2A REF= stOs[iVoltaDoComando.dwLowPart].Sa.xObjPresente;
		
										3:
											RefIT3A REF= stOs[iVoltaDoComando.dwLowPart].Sa.xObjPresente;
		
										4:
											RefIT4A REF= stOs[iVoltaDoComando.dwLowPart].Sa.xObjPresente;
									END_CASE
		
									iTag := iTag + 1;
								END_IF
							END_IF
						END_IF
					ELSE
						FOR i := DINT_TO_INT(LOWER_BOUND(stOutros, 1)) TO DINT_TO_INT(UPPER_BOUND(stOutros, 1)) DO
							IF stOutros[i].sTag = sTag1[iTag] THEN
								CASE iTag OF
									1:
										RefIT1A REF= stOutros[i].xEstado;
	
									2:
										RefIT2A REF= stOutros[i].xEstado;
	
									3:
										RefIT3A REF= stOutros[i].xEstado;
	
									4:
										RefIT4A REF= stOutros[i].xEstado;
								END_CASE
	
								iTag := iTag + 1;
								EXIT;
							END_IF
						END_FOR
					END_IF
				END_IF
			ELSE
				iTag := iTag + 1;
			END_IF
		ELSE
			CASE iTag OF
				1:
					RefIT1A REF= Falso;

				2:
					RefIT2A REF= Falso;

				3:
					RefIT3A REF= Falso;

				4:
					RefIT4A REF= Falso;
			END_CASE

			iTag := iTag + 1;
		END_IF

		
		
		
		
	enum_MaquinaConfigPartidaDB.ProcuraTag2:
		IF sTag2[iTag] <> '' THEN
			CASE iTag OF
				1:
					xDiferenteDoAnterior := sTag2[iTag] <> EstruturaAnterior.IT1B;
	
				2:
					xDiferenteDoAnterior := sTag2[iTag] <> EstruturaAnterior.IT2B;
	
				3:
					xDiferenteDoAnterior := sTag2[iTag] <> EstruturaAnterior.IT3B;
	
				4:
					xDiferenteDoAnterior := sTag2[iTag] <> EstruturaAnterior.IT4B;
			END_CASE
		
		
			IF xDiferenteDoAnterior THEN
				IF FIND(STR1 := sTag2[iTag], STR2 := 'M') = 1 THEN
	
					TagAProcurar		:= sTag2[iTag];
					stPara.eParaType	:= E_ExpParameterType.STRING_;
					stPara.nParaSize	:= SIZEOF(TagAProcurar);
					stPara.sParaName	:= 'Tag';
	
					// set command with placeholder
					sCmd := CONCAT(CONCAT(CONCAT(CONCAT('SELECT motor FROM geral.',sNomeDataBase),' where Tag=$''), TagAProcurar), '$';');
	
					// call functionblock
					IF NOT xNaoAtualiza THEN
						IF fbPLCDBCmd.ExecuteDataReturn
							(
								hDBID := 1,
									pExpression := ADR(sCmd),
									cbExpression := SIZEOF(sCmd),
									pData := ADR(TagAProcurar),
									cbData := SIZEOF(TagAProcurar),
									pParameter := ADR(stPara),
									cbParameter := SIZEOF(stPara),
									nStartIndex := 0,
									nRecordCount := 1,
									pReturnData := ADR(iVoltaDoComando),
									cbReturnData := SIZEOF(iVoltaDoComando),
									pRecords := ADR(nRecords))
						THEN
							IF fbPLCDBCmd.bError THEN
								sMensagemErro1 := 'Nao conseguiu a tag';
								{error <'Não conseguiu ler TAG2A no banco no bloco FB_ConfigPartidaNoBanco 7'>}
							ELSE
								sMensagemErro1 := 'Conseguiu a tag';
		
								CASE iTag OF
									1:
										RefIT1B REF= stMotor[iVoltaDoComando.dwLowPart].Sa.xNaoLigaProxMotor;
		
									2:
										RefIT2B REF= stMotor[iVoltaDoComando.dwLowPart].Sa.xNaoLigaProxMotor;
		
									3:
										RefIT3B REF= stMotor[iVoltaDoComando.dwLowPart].Sa.xNaoLigaProxMotor;
		
									4:
										RefIT4B REF= stMotor[iVoltaDoComando.dwLowPart].Sa.xNaoLigaProxMotor;
								END_CASE
		
								iTag := iTag + 1;
							END_IF
						END_IF
					END_IF
				ELSE
					IF FIND(STR1 := sTag2[iTag], STR2 := 'S') = 1 THEN
						//quando for sensor
						TagAProcurar		:= sTag2[iTag];
						stPara.eParaType	:= E_ExpParameterType.STRING_;
						stPara.nParaSize	:= SIZEOF(TagAProcurar);
						stPara.sParaName	:= 'Tag';
	
						// set command with placeholder
						sCmd := CONCAT(CONCAT('SELECT sensor FROM geral.sensoresconfig where Tag=$'', TagAProcurar), '$';');
	
						// call functionblock
						IF NOT xNaoAtualiza THEN
							IF fbPLCDBCmd.ExecuteDataReturn
								(
									hDBID := 1,
										pExpression := ADR(sCmd),
										cbExpression := SIZEOF(sCmd),
										pData := ADR(TagAProcurar),
										cbData := SIZEOF(TagAProcurar),
										pParameter := ADR(stPara),
										cbParameter := SIZEOF(stPara),
										nStartIndex := 0,
										nRecordCount := 1,
										pReturnData := ADR(iVoltaDoComando),
										cbReturnData := SIZEOF(iVoltaDoComando),
										pRecords := ADR(nRecords))
							THEN
								IF fbPLCDBCmd.bError THEN
									sMensagemErro1 := 'Nao conseguiu a tag';
									{error <'Não conseguiu ler TAG2B no banco no bloco FB_ConfigPartidaNoBanco 8'>}
								ELSE
									sMensagemErro1 := 'Conseguiu a tag';
		
									CASE iTag OF
										1:
											RefIT1B REF= stSensores[iVoltaDoComando.dwLowPart].Sa.xObjPresente;
		
										2:
											RefIT2B REF= stSensores[iVoltaDoComando.dwLowPart].Sa.xObjPresente;
		
										3:
											RefIT3B REF= stSensores[iVoltaDoComando.dwLowPart].Sa.xObjPresente;
		
										4:
											RefIT4B REF= stSensores[iVoltaDoComando.dwLowPart].Sa.xObjPresente;
									END_CASE
		
									iTag := iTag + 1;
								END_IF
							END_IF
						END_IF
					ELSIF FIND(STR1 := sTag2[iTag], STR2 := 'OE') = 1 THEN
						//quando for sensor
						TagAProcurar		:= sTag2[iTag];
						stPara.eParaType	:= E_ExpParameterType.STRING_;
						stPara.nParaSize	:= SIZEOF(TagAProcurar);
						stPara.sParaName	:= 'Tag';
	
						// set command with placeholder
						sCmd := CONCAT(CONCAT('SELECT sensor FROM geral.oeconfig where Tag=$'', TagAProcurar), '$';');
	
						// call functionblock
						IF NOT xNaoAtualiza THEN
							IF fbPLCDBCmd.ExecuteDataReturn
								(
									hDBID := 1,
										pExpression := ADR(sCmd),
										cbExpression := SIZEOF(sCmd),
										pData := ADR(TagAProcurar),
										cbData := SIZEOF(TagAProcurar),
										pParameter := ADR(stPara),
										cbParameter := SIZEOF(stPara),
										nStartIndex := 0,
										nRecordCount := 1,
										pReturnData := ADR(iVoltaDoComando),
										cbReturnData := SIZEOF(iVoltaDoComando),
										pRecords := ADR(nRecords))
							THEN
								IF fbPLCDBCmd.bError THEN
									sMensagemErro1 := 'Nao conseguiu a tag';
									{error <'Não conseguiu ler TAG2B no banco no bloco FB_ConfigPartidaNoBanco 8'>}
								ELSE
									sMensagemErro1 := 'Conseguiu a tag';
		
									CASE iTag OF
										1:
											RefIT1B REF= stOe[iVoltaDoComando.dwLowPart].Sa.xObjPresente;
		
										2:
											RefIT2B REF= stOe[iVoltaDoComando.dwLowPart].Sa.xObjPresente;
		
										3:
											RefIT3B REF= stOe[iVoltaDoComando.dwLowPart].Sa.xObjPresente;
		
										4:
											RefIT4B REF= stOe[iVoltaDoComando.dwLowPart].Sa.xObjPresente;
									END_CASE
		
									iTag := iTag + 1;
								END_IF
							END_IF
						END_IF
					ELSIF FIND(STR1 := sTag2[iTag], STR2 := 'OS') = 1 THEN
						//quando for sensor
						TagAProcurar		:= sTag2[iTag];
						stPara.eParaType	:= E_ExpParameterType.STRING_;
						stPara.nParaSize	:= SIZEOF(TagAProcurar);
						stPara.sParaName	:= 'Tag';
	
						// set command with placeholder
						sCmd := CONCAT(CONCAT('SELECT sensor FROM geral.osconfig where Tag=$'', TagAProcurar), '$';');
	
						// call functionblock
						IF NOT xNaoAtualiza THEN
							IF fbPLCDBCmd.ExecuteDataReturn
								(
									hDBID := 1,
										pExpression := ADR(sCmd),
										cbExpression := SIZEOF(sCmd),
										pData := ADR(TagAProcurar),
										cbData := SIZEOF(TagAProcurar),
										pParameter := ADR(stPara),
										cbParameter := SIZEOF(stPara),
										nStartIndex := 0,
										nRecordCount := 1,
										pReturnData := ADR(iVoltaDoComando),
										cbReturnData := SIZEOF(iVoltaDoComando),
										pRecords := ADR(nRecords))
							THEN
								IF fbPLCDBCmd.bError THEN
									sMensagemErro1 := 'Nao conseguiu a tag';
									{error <'Não conseguiu ler TAG2B no banco no bloco FB_ConfigPartidaNoBanco 8'>}
								ELSE
									sMensagemErro1 := 'Conseguiu a tag';
		
									CASE iTag OF
										1:
											RefIT1B REF= stOs[iVoltaDoComando.dwLowPart].Sa.xObjPresente;
		
										2:
											RefIT2B REF= stOs[iVoltaDoComando.dwLowPart].Sa.xObjPresente;
		
										3:
											RefIT3B REF= stOs[iVoltaDoComando.dwLowPart].Sa.xObjPresente;
		
										4:
											RefIT4B REF= stOs[iVoltaDoComando.dwLowPart].Sa.xObjPresente;
									END_CASE
		
									iTag := iTag + 1;
								END_IF
							END_IF
						END_IF
					ELSE
						FOR i := DINT_TO_INT(LOWER_BOUND(stOutros, 1)) TO DINT_TO_INT(UPPER_BOUND(stOutros, 1)) DO
							IF stOutros[i].sTag = sTag2[iTag] THEN
								CASE iTag OF
									1:
										RefIT1B REF= stOutros[i].xEstado;
	
									2:
										RefIT2B REF= stOutros[i].xEstado;
	
									3:
										RefIT3B REF= stOutros[i].xEstado;
	
									4:
										RefIT4B REF= stOutros[i].xEstado;
								END_CASE
	
								iTag := iTag + 1;
								EXIT;
							END_IF
						END_FOR
					END_IF
				END_IF
			ELSE
				iTag := iTag + 1;
			END_IF
		ELSE
			CASE iTag OF
				1:
					RefIT1B REF= Falso;

				2:
					RefIT2B REF= Falso;

				3:
					RefIT3B REF= Falso;

				4:
					RefIT4B REF= Falso;
			END_CASE

			iTag := iTag + 1;
		END_IF

	enum_MaquinaConfigPartidaDB.Gera_sInterlock:
		iAux := iAux;

